TYPE "UDT_RIOVSUStatus"
VERSION : 0.1
   STRUCT
      PNSlaveNotOnline { ExternalAccessible := 'False'; ExternalVisible := 'False'; ExternalWritable := 'False'} : Bool;   // Profinet slave is not online
      PNSlaveError { ExternalAccessible := 'False'; ExternalVisible := 'False'; ExternalWritable := 'False'} : Bool;   // Profinet slave has an error
      "400VCircuitBreaker" { ExternalAccessible := 'False'; ExternalVisible := 'False'; ExternalWritable := 'False'} : Bool;   // 400V Circuit breaker has tripped
      BrakeCircuitBreaker { ExternalAccessible := 'False'; ExternalVisible := 'False'; ExternalWritable := 'False'} : Bool;   // Brake Circuit breaker has tripped
      BrakeThermalError { ExternalAccessible := 'False'; ExternalVisible := 'False'; ExternalWritable := 'False'} : Bool;   // Brake of the servo unit is giving a thermal error
      "24VPowersupplyError" { ExternalAccessible := 'False'; ExternalVisible := 'False'; ExternalWritable := 'False'} : Bool;   // 24V power supply is in error
      ET200sp_ErrorModule : Array[0..31] of Bool;   // True = ET200sp Module has an error or is offline
      PNSlaveWarning { ExternalAccessible := 'False'; ExternalVisible := 'False'; ExternalWritable := 'False'} : Bool;   // Profinet slave has a warning
   END_STRUCT;

END_TYPE

TYPE "UDT_VSUInterface"
TITLE = UDT_VSUInterface
VERSION : 0.1
//User-defined structure of VSU interface parameters.
   STRUCT
      Decisionpoint : Int;   // Point in tracking where the destination is found on the VSU conveyor [mm]
      RequestedPosition : Int;   // Position Requested by destination block
      PositionSetpoint : Int;   // Position number (as configured) to go to by positioning device
      PositionActual : Int;   // Position number the positioning device is actually on
      SwitchingTime : UInt;   // Time it takes to go from one position to the next [ms]
      VSUMainPowerOk { ExternalAccessible := 'False'; ExternalVisible := 'False'; ExternalWritable := 'False'} : Bool;   // True = Main power for VSU ok
      BrakeOk { ExternalAccessible := 'False'; ExternalVisible := 'False'; ExternalWritable := 'False'} : Bool;   // True = VSU brake is ok
      PNDeviceOk { ExternalAccessible := 'False'; ExternalVisible := 'False'; ExternalWritable := 'False'} : Bool;   // Device ok
      Automatic { ExternalAccessible := 'False'; ExternalVisible := 'False'; ExternalWritable := 'False'} : Bool;   // Automatic mode request
      RunEnabled { ExternalAccessible := 'False'; ExternalVisible := 'False'; ExternalWritable := 'False'} : Bool;   // Running of the positioning device is enabled by VSU
      GoReference { ExternalAccessible := 'False'; ExternalVisible := 'False'; ExternalWritable := 'False'} : Bool;   // Activate reference run by VSU
      Referenced { ExternalAccessible := 'False'; ExternalVisible := 'False'; ExternalWritable := 'False'} : Bool;   // Positioning device is referenced
      Manual { ExternalAccessible := 'False'; ExternalVisible := 'False'; ExternalWritable := 'False'} : Bool;   // Manual mode request
      Reference_command { ExternalAccessible := 'False'; ExternalVisible := 'False'; ExternalWritable := 'False'} : Bool;   // Refference command
      JogUp { ExternalAccessible := 'False'; ExternalVisible := 'False'; ExternalWritable := 'False'} : Bool;   // Jog request to move equipment up
      JogDown { ExternalAccessible := 'False'; ExternalVisible := 'False'; ExternalWritable := 'False'} : Bool;   // Jog request to move equipment down
      Ready { ExternalAccessible := 'False'; ExternalVisible := 'False'; ExternalWritable := 'False'} : Bool;   // Positioning block is running and error free
      MotorRunning { ExternalAccessible := 'False'; ExternalVisible := 'False'; ExternalWritable := 'False'} : Bool;   // Motor is running
      Positioning { ExternalAccessible := 'False'; ExternalVisible := 'False'; ExternalWritable := 'False'} : Bool;   // positioning device is moving to its position
      ResetStatistics { ExternalAccessible := 'False'; ExternalVisible := 'False'; ExternalWritable := 'False'} : Bool;   // Reset statistics
      InternalErrorRIOPanel { ExternalAccessible := 'False'; ExternalVisible := 'False'; ExternalWritable := 'False'} : Bool;   // RIO panel has an internal error
      InternalWarningRIOPanel { ExternalAccessible := 'False'; ExternalVisible := 'False'; ExternalWritable := 'False'} : Bool;   // RIO panel has an internal waring
      InternalErrorVFD { ExternalAccessible := 'False'; ExternalVisible := 'False'; ExternalWritable := 'False'} : Bool;   // positioning device internal error
      InternalWarningVFD { ExternalAccessible := 'False'; ExternalVisible := 'False'; ExternalWritable := 'False'} : Bool;   // positioning device has a warning
      InternalErrorReset { ExternalAccessible := 'False'; ExternalVisible := 'False'; ExternalWritable := 'False'} : Bool;   // Reset internal faults
      StartLowSpeed { ExternalAccessible := 'False'; ExternalVisible := 'False'; ExternalWritable := 'False'} : Bool;   // Positioning device starting in low speed
      RequestDieBackUpstream { ExternalAccessible := 'False'; ExternalVisible := 'False'; ExternalWritable := 'False'} : Bool;   // External request die back to the upstream conveyor of the VSU
      ExternalHold { ExternalAccessible := 'False'; ExternalVisible := 'False'; ExternalWritable := 'False'} : Bool;   // External request to stop the VSU conveyor
   END_STRUCT;

END_TYPE

TYPE "UDT_VfdPositioningStatus"
TITLE = UDT_VfdPositioningStatus
VERSION : 0.1
//User-defined structure of VFD SEW positioning status.
   STRUCT
      ErrorCode : Int;   // Error code
      SubErrorCode : Int;   // Sub error code
      PNSlaveNotOnline : Bool := FALSE;   // Profinet slave is not on line
      PNSlaveError : Bool := FALSE;   // Profinet slave has an error
      InternalError : Bool := FALSE;   // A VFD internal error is active, see error code
      InternalWarning : Bool := FALSE;   // A VFD internal warning is active, see error code
      CommunicationErrorMovikit : Bool := FALSE;   // Communication error with MoviKit
      PositioningTimeOutError : Bool := FALSE;   // Exceeded time to reach position
      PNSlaveWarning { ExternalAccessible := 'False'; ExternalVisible := 'False'; ExternalWritable := 'False'} : Bool;   // Profinet slave has a warning
   END_STRUCT;

END_TYPE

TYPE "UDT_VSULiftStatistics"
TITLE = UDT_VSUStatistics
VERSION : 0.1
//User-defined structure of FB_VerticalSwitch function block statistics.
   STRUCT
      UpTime { ExternalWritable := 'False'} : "UDT_EventStatistic";   // VSU up time
      DownTime { ExternalWritable := 'False'} : "UDT_EventStatistic";   // VSU down time
      ExitGapErr { ExternalWritable := 'False'} : "UDT_EventStatistic";   // Error statistics for VSU
      EntryGapErr { ExternalWritable := 'False'} : "UDT_EventStatistic";   // Error statistics for VSU
      BeltTear1Err { ExternalWritable := 'False'} : "UDT_EventStatistic";   // Error statistics for VSU
      BeltTear2Err { ExternalWritable := 'False'} : "UDT_EventStatistic";   // Error statistics for VSU
      MaintSupport1Err { ExternalWritable := 'False'} : "UDT_EventStatistic";   // Error statistics for VSU
      MaintSupport2Err { ExternalWritable := 'False'} : "UDT_EventStatistic";   // Error statistics for VSU
      UpperPositionErr { ExternalWritable := 'False'} : "UDT_EventStatistic";   // Error statistics for VSU
      LowerPositionErr { ExternalWritable := 'False'} : "UDT_EventStatistic";   // Error statistics for VSU
      SafetyDoorErr { ExternalWritable := 'False'} : "UDT_EventStatistic";   // Error statistics for VSU
      Direction_Error { ExternalWritable := 'False'} : "UDT_EventStatistic";   // Error statistics for VSU
   END_STRUCT;

END_TYPE

TYPE "UDT_VfdPositioningConfiguration"
TITLE = UDT_VfdPositioningConfiguration
VERSION : 0.1
//User defined stucture for configuring positioning device
   STRUCT
      TorqueMax : Real;   // VFD torque max - reference [Nm] as set up in SEW project
      SupplyFdbckOnDelayTime : UDInt;   // On delay time for supply feedback [ms]
      PositionWindow : DInt;   // Position window (tolerance) [mm]
      PositionMax : DInt;   // Maximum allowed position [mm]
      PositionMin : DInt;   // Minimum allowed position [mm]
      VFDSpeed : Int;   // Speed to run in automatic mode [mm/s]
      VFDAccDecel : Int;   // Acceleration and deceleration [mm/s2]
      VFDPNDeviceName : String;   // VFD's device name
      Position : Array[0..10] of DInt;   // Positions in mm to move to as requested
   END_STRUCT;

END_TYPE

TYPE "UDT_VfdSEWSpeedPO"
TITLE = UDT_VFD_SEW_PO
VERSION : 0.1
//User-defined structure of VFD SEW output telegram.
   STRUCT
      Control_Word_1 : Struct   // Control Word 1
         ResetError { ExternalAccessible := 'False'; ExternalVisible := 'False'; ExternalWritable := 'False'} : Bool;   // Reset error "1"
         BIT_09_Reserved { ExternalAccessible := 'False'; ExternalVisible := 'False'; ExternalWritable := 'False'} : Bool;   // Reserved
         ActivateDriveTrain2 { ExternalAccessible := 'False'; ExternalVisible := 'False'; ExternalWritable := 'False'} : Bool;   // Activate drive train 2 "1"
         BIT_11_Reserved { ExternalAccessible := 'False'; ExternalVisible := 'False'; ExternalWritable := 'False'} : Bool;   // Reserved
         DeactivateSW_LimitSwitch { ExternalAccessible := 'False'; ExternalVisible := 'False'; ExternalWritable := 'False'} : Bool;   // Deactivate software limit switch "1"
         ActivateInhibit { ExternalAccessible := 'False'; ExternalVisible := 'False'; ExternalWritable := 'False'} : Bool;   // Activate inhibit "1"
         ActivateStandby { ExternalAccessible := 'False'; ExternalVisible := 'False'; ExternalWritable := 'False'} : Bool;   // Activate standby "1"
         MovikitHandshakeIn { ExternalAccessible := 'False'; ExternalVisible := 'False'; ExternalWritable := 'False'} : Bool;   // If the MOVIKIT works the value will be copied into "MovikitHandshakeOut"
         EnableRapidStop { ExternalAccessible := 'False'; ExternalVisible := 'False'; ExternalWritable := 'False'} : Bool;   // Enable “1” / Rapid stop “0”
         EnableApplicationStop { ExternalAccessible := 'False'; ExternalVisible := 'False'; ExternalWritable := 'False'} : Bool;   // Enable “1” / Application stop “0”
         BIT_02_Reserved { ExternalAccessible := 'False'; ExternalVisible := 'False'; ExternalWritable := 'False'} : Bool;   // Reserved
         ReleaseBrake { ExternalAccessible := 'False'; ExternalVisible := 'False'; ExternalWritable := 'False'} : Bool;   // Release brake "1"
         JogPos { ExternalAccessible := 'False'; ExternalVisible := 'False'; ExternalWritable := 'False'} : Bool;   // Jog in positive direction "1"
         JogNeg { ExternalAccessible := 'False'; ExternalVisible := 'False'; ExternalWritable := 'False'} : Bool;   // Jog in negative direction "1"
         ApplyRelativePositioning { ExternalAccessible := 'False'; ExternalVisible := 'False'; ExternalWritable := 'False'} : Bool;   // Take the relative position from the FCB09 "1"
         StartStop { ExternalAccessible := 'False'; ExternalVisible := 'False'; ExternalWritable := 'False'} : Bool;   // Start "1" / Stop "0"
      END_STRUCT;
      SetpointSpeed : Int;   // Speed (Int) in rpm
      SetpointAcceleration : Int;   // Acceleration (Int) in rpm/s
      SetpointDeceleration : Int;   // Decceleration (Int) in rpm/s
   END_STRUCT;

END_TYPE

TYPE "UDT_AixPlcFullControllerConfiguration"
TITLE = UDT_VFD_Configuration
VERSION : 0.1
//User-defined structure oparameters.
   STRUCT
      AixContrlPNDeviceName { ExternalAccessible := 'False'; ExternalVisible := 'False'; ExternalWritable := 'False'} : String;   // Ai2's Controller Profinet device name
      Motor { ExternalAccessible := 'False'; ExternalVisible := 'False'; ExternalWritable := 'False'} : Struct
         RampUpTime { ExternalAccessible := 'False'; ExternalVisible := 'False'; ExternalWritable := 'False'} : UDInt := 100;   // Ramp up time for monitoring starting [ms]
         RampDownTime { ExternalAccessible := 'False'; ExternalVisible := 'False'; ExternalWritable := 'False'} : UDInt := 100;   // Ramp up time for monitoring stopping [ms]
         SpeedSetpointWindow { ExternalAccessible := 'False'; ExternalVisible := 'False'; ExternalWritable := 'False'} : Int := 5;   // Speed setpoint window (tolerance) [mm/s]
         Ratio { ExternalAccessible := 'False'; ExternalVisible := 'False'; ExternalWritable := 'False'} : Real := 1.0;   // Ratio conveyor roller to driven roller
         DirectionReversal { ExternalAccessible := 'False'; ExternalVisible := 'False'; ExternalWritable := 'False'} : Bool;   // True = direction will be reversed
         InterlockFwd { ExternalAccessible := 'False'; ExternalVisible := 'False'; ExternalWritable := 'False'} : Bool := TRUE;   // False = running in forward direction is not possible / allowed
         InterlockRvs { ExternalAccessible := 'False'; ExternalVisible := 'False'; ExternalWritable := 'False'} : Bool;   // False = running in reverse direction is not possible / allowed
         MotorExist { ExternalAccessible := 'False'; ExternalVisible := 'False'; ExternalWritable := 'False'} : Bool;   // True = Motor output connected
      END_STRUCT;
   END_STRUCT;

END_TYPE

TYPE "UDT_AixPlcFullIn"
VERSION : 0.1
   STRUCT
      ConveyStopStatus { ExternalVisible := 'False'} : Struct   // Status of ConveyStop
         Bit08 { ExternalAccessible := 'False'; ExternalVisible := 'False'; ExternalWritable := 'False'} : Bool;   // Reserved
         Bit09 { ExternalAccessible := 'False'; ExternalVisible := 'False'; ExternalWritable := 'False'} : Bool;   // Reserved
         StopActiveCommandPLC { ExternalAccessible := 'False'; ExternalVisible := 'False'; ExternalWritable := 'False'} : Bool;   // Stop active due to stop command from the PLC
         Bit11 { ExternalAccessible := 'False'; ExternalVisible := 'False'; ExternalWritable := 'False'} : Bool;   // Reserved
         Bit12 { ExternalAccessible := 'False'; ExternalVisible := 'False'; ExternalWritable := 'False'} : Bool;   // Reserved
         Bit13 { ExternalAccessible := 'False'; ExternalVisible := 'False'; ExternalWritable := 'False'} : Bool;   // Reserved
         Bit14 { ExternalAccessible := 'False'; ExternalVisible := 'False'; ExternalWritable := 'False'} : Bool;   // Reserved
         Bit15 { ExternalAccessible := 'False'; ExternalVisible := 'False'; ExternalWritable := 'False'} : Bool;   // Reserved
         Bit00 { ExternalAccessible := 'False'; ExternalVisible := 'False'; ExternalWritable := 'False'} : Bool;   // Reserved
         Bit01 { ExternalAccessible := 'False'; ExternalVisible := 'False'; ExternalWritable := 'False'} : Bool;   // Reserved
         Bit02 { ExternalAccessible := 'False'; ExternalVisible := 'False'; ExternalWritable := 'False'} : Bool;   // Reserved
         Bit03 { ExternalAccessible := 'False'; ExternalVisible := 'False'; ExternalWritable := 'False'} : Bool;   // Reserved
         Bit04 { ExternalAccessible := 'False'; ExternalVisible := 'False'; ExternalWritable := 'False'} : Bool;   // Reserved
         StopActiveOtherModule { ExternalAccessible := 'False'; ExternalVisible := 'False'; ExternalWritable := 'False'} : Bool;   // Stop condition is active on a module in the ConveyStop group
         StopActiveLostConn { ExternalAccessible := 'False'; ExternalVisible := 'False'; ExternalWritable := 'False'} : Bool;   // Stop is active due to a loss of communication connection
         StopActiveLostPLC { ExternalAccessible := 'False'; ExternalVisible := 'False'; ExternalWritable := 'False'} : Bool;   // Stop active due to a loss of connection with the PLC
      END_STRUCT;
      AllSensorPortInputs { ExternalVisible := 'False'} : Struct   // Left and Right Sensor Port inputs
         Bit08 { ExternalAccessible := 'False'; ExternalVisible := 'False'; ExternalWritable := 'False'} : Bool;   // Reserved
         Bit09 { ExternalAccessible := 'False'; ExternalVisible := 'False'; ExternalWritable := 'False'} : Bool;   // Reserved
         Bit10 { ExternalAccessible := 'False'; ExternalVisible := 'False'; ExternalWritable := 'False'} : Bool;   // Reserved
         Bit11 { ExternalAccessible := 'False'; ExternalVisible := 'False'; ExternalWritable := 'False'} : Bool;   // Reserved
         Bit12 { ExternalAccessible := 'False'; ExternalVisible := 'False'; ExternalWritable := 'False'} : Bool;   // Reserved
         Bit13 { ExternalAccessible := 'False'; ExternalVisible := 'False'; ExternalWritable := 'False'} : Bool;   // Reserved
         Bit14 { ExternalAccessible := 'False'; ExternalVisible := 'False'; ExternalWritable := 'False'} : Bool;   // Reserved
         Heartbeat { ExternalAccessible := 'False'; ExternalVisible := 'False'; ExternalWritable := 'False'} : Bool;   // This bit toggles every 2 seconds
         LeftPin2 { ExternalAccessible := 'False'; ExternalVisible := 'False'; ExternalWritable := 'False'} : Bool;   // Left sensor port Pin2 state
         Bit01 { ExternalAccessible := 'False'; ExternalVisible := 'False'; ExternalWritable := 'False'} : Bool;   // Reserved
         RightPin2 { ExternalAccessible := 'False'; ExternalVisible := 'False'; ExternalWritable := 'False'} : Bool;   // Right sensor port Pin2 state
         Bit03 { ExternalAccessible := 'False'; ExternalVisible := 'False'; ExternalWritable := 'False'} : Bool;   // Reserved
         LeftSensor { ExternalAccessible := 'False'; ExternalVisible := 'False'; ExternalWritable := 'False'} : Bool;   // Left sensor port Pin4 state
         Bit05 { ExternalAccessible := 'False'; ExternalVisible := 'False'; ExternalWritable := 'False'} : Bool;   // Reserved
         RightSensor { ExternalAccessible := 'False'; ExternalVisible := 'False'; ExternalWritable := 'False'} : Bool;   // Right sensor port Pin4 state
         Bit07 { ExternalAccessible := 'False'; ExternalVisible := 'False'; ExternalWritable := 'False'} : Bool;   // Reserved
      END_STRUCT;
      SensorDetect { ExternalVisible := 'False'} : Struct   // Sensor detection
         Bits08_15 { ExternalVisible := 'False'} : SInt;   // Reserved
         RightSensorDetect { ExternalAccessible := 'False'; ExternalVisible := 'False'; ExternalWritable := 'False'} : Bool;   // True when sensor is detected
         LeftSensorDetect { ExternalAccessible := 'False'; ExternalVisible := 'False'; ExternalWritable := 'False'} : Bool;   // True when sensor is detected
         Bit02 { ExternalAccessible := 'False'; ExternalVisible := 'False'; ExternalWritable := 'False'} : Bool;   // Reserved
         Bit03 { ExternalAccessible := 'False'; ExternalVisible := 'False'; ExternalWritable := 'False'} : Bool;   // Reserved
         Bit04 { ExternalAccessible := 'False'; ExternalVisible := 'False'; ExternalWritable := 'False'} : Bool;   // Reserved
         Bit05 { ExternalAccessible := 'False'; ExternalVisible := 'False'; ExternalWritable := 'False'} : Bool;   // Reserved
         Bit06 { ExternalAccessible := 'False'; ExternalVisible := 'False'; ExternalWritable := 'False'} : Bool;   // Reserved
         Bit07 { ExternalAccessible := 'False'; ExternalVisible := 'False'; ExternalWritable := 'False'} : Bool;   // Reserved
      END_STRUCT;
      VoltageMotors { ExternalVisible := 'False'} : Int;   // The Voltage applied to the module's motor power connection in millivolts
      LeftMotorCurrent { ExternalVisible := 'False'} : Int;   // Left motor running current in milliamperes
      LeftMotorFreq { ExternalVisible := 'False'} : Int;   // Left motor running electrical frequency in Hz
      LeftMotorCalcTemp { ExternalVisible := 'False'} : Byte;   // Left motor temperature in degrees C
      ModuleTemp { ExternalVisible := 'False'} : Byte;   // Module CPU temperature in degrees C
      LeftMotorDiagnostic { ExternalVisible := 'False'} : Struct   // Left motor diagnostics .
         Overheat { ExternalAccessible := 'False'; ExternalVisible := 'False'; ExternalWritable := 'False'} : Bool;   // Left motor temperature has exceeded 105 degrees Celsius
         MaxTorque { ExternalAccessible := 'False'; ExternalVisible := 'False'; ExternalWritable := 'False'} : Bool;   // Left motor at maximum torque output
         ShortCircuit { ExternalAccessible := 'False'; ExternalVisible := 'False'; ExternalWritable := 'False'} : Bool;   // Left motor short circuit
         MotorNotConnected { ExternalAccessible := 'False'; ExternalVisible := 'False'; ExternalWritable := 'False'} : Bool;   // Left motor is not connected
         Overload { ExternalAccessible := 'False'; ExternalVisible := 'False'; ExternalWritable := 'False'} : Bool;   // Left motor overloaded after more than 20 seconds in Stalled
         Stalled { ExternalAccessible := 'False'; ExternalVisible := 'False'; ExternalWritable := 'False'} : Bool;   // Left motor stalled and speed is less than 10% of the set speed
         BadHall { ExternalAccessible := 'False'; ExternalVisible := 'False'; ExternalWritable := 'False'} : Bool;   // Left motor Hall Effect Sensor error active
         MotorNotUsed { ExternalAccessible := 'False'; ExternalVisible := 'False'; ExternalWritable := 'False'} : Bool;   // Left motor not used
         MotorStatus1 { ExternalAccessible := 'False'; ExternalVisible := 'False'; ExternalWritable := 'False'} : Bool;   // Left motor running and direction status
         MotorStatus2 { ExternalAccessible := 'False'; ExternalVisible := 'False'; ExternalWritable := 'False'} : Bool;   // Left motor running and direction status
         MotorPortinDOmode { ExternalAccessible := 'False'; ExternalVisible := 'False'; ExternalWritable := 'False'} : Bool;   // Left motor port is in digital Output mode .
         ReservedBit03 { ExternalAccessible := 'False'; ExternalVisible := 'False'; ExternalWritable := 'False'} : Bool;   // Reserved
         ReservedBit04 { ExternalAccessible := 'False'; ExternalVisible := 'False'; ExternalWritable := 'False'} : Bool;   // Reserved
         BoardOverheat { ExternalAccessible := 'False'; ExternalVisible := 'False'; ExternalWritable := 'False'} : Bool;   // Board temperature has exceeded 90 degrees Celsius
         OverVoltage { ExternalAccessible := 'False'; ExternalVisible := 'False'; ExternalWritable := 'False'} : Bool;   // Supply voltage + motor back EMF exceeded 30 volts
         LowVoltage { ExternalAccessible := 'False'; ExternalVisible := 'False'; ExternalWritable := 'False'} : Bool;   // Module power supply is less than 18 Volts
      END_STRUCT;
      RightMotorCurrent { ExternalVisible := 'False'} : Int;   // Right motor running current in milliamperes
      RightMotorFreq { ExternalVisible := 'False'} : Int;   // Right motor running electrical frequency in Hz
      RightMotorCalcTemp { ExternalVisible := 'False'} : Byte;   // Right motor temperature in degrees Celsius
      ModuleTemp1 { ExternalVisible := 'False'} : Byte;   // Module PCB temperature in degrees C (same as ModuleTemp tag)
      RightMotorDiagnostic { ExternalVisible := 'False'} : Struct   // Right motor diagnostics .
         Overheat { ExternalAccessible := 'False'; ExternalVisible := 'False'; ExternalWritable := 'False'} : Bool;   // Right motor temperature has exceeded 105 degrees Celsius
         MaxTorque { ExternalAccessible := 'False'; ExternalVisible := 'False'; ExternalWritable := 'False'} : Bool;   // Right motor at maximum torque output
         ShortCircuit { ExternalAccessible := 'False'; ExternalVisible := 'False'; ExternalWritable := 'False'} : Bool;   // Right motor short circuit
         MotorNotConnected { ExternalAccessible := 'False'; ExternalVisible := 'False'; ExternalWritable := 'False'} : Bool;   // Right motor is not connected
         Overload { ExternalAccessible := 'False'; ExternalVisible := 'False'; ExternalWritable := 'False'} : Bool;   // Right motor overloaded after more than 20 seconds in Stalled
         Stalled { ExternalAccessible := 'False'; ExternalVisible := 'False'; ExternalWritable := 'False'} : Bool;   // Right motor stalled and speed is less than 10% of the set speed
         BadHall { ExternalAccessible := 'False'; ExternalVisible := 'False'; ExternalWritable := 'False'} : Bool;   // Right motor Hall Effect Sensor error active
         MotorNotUsed { ExternalAccessible := 'False'; ExternalVisible := 'False'; ExternalWritable := 'False'} : Bool;   // Right motor is not used
         MotorStatus1 { ExternalAccessible := 'False'; ExternalVisible := 'False'; ExternalWritable := 'False'} : Bool;   // Right motor running and direction status
         MotorStatus2 { ExternalAccessible := 'False'; ExternalVisible := 'False'; ExternalWritable := 'False'} : Bool;   // Right motor running and direction status
         MotorPortinDOmode { ExternalAccessible := 'False'; ExternalVisible := 'False'; ExternalWritable := 'False'} : Bool;   // Right motor port is in digital output mode .
         ReservedBit03 { ExternalAccessible := 'False'; ExternalVisible := 'False'; ExternalWritable := 'False'} : Bool;   // Reserved
         ReservedBit04 { ExternalAccessible := 'False'; ExternalVisible := 'False'; ExternalWritable := 'False'} : Bool;   // Reserved
         BoardOverheat { ExternalAccessible := 'False'; ExternalVisible := 'False'; ExternalWritable := 'False'} : Bool;   // Board temperature has exceeded 90 degrees Celsius
         OverVoltage { ExternalAccessible := 'False'; ExternalVisible := 'False'; ExternalWritable := 'False'} : Bool;   // Supply voltage + motor back EMF exceeded 30 volts
         LowVoltage { ExternalAccessible := 'False'; ExternalVisible := 'False'; ExternalWritable := 'False'} : Bool;   // Module power supply is less than 18 Volts
      END_STRUCT;
      LeftMotorDIOstatus { ExternalVisible := 'False'} : Struct   // Status of Left M8 motor port when used as a digital IO
         Bit08 { ExternalAccessible := 'False'; ExternalVisible := 'False'; ExternalWritable := 'False'} : Bool;   // Reserved
         Bit09 { ExternalAccessible := 'False'; ExternalVisible := 'False'; ExternalWritable := 'False'} : Bool;   // Reserved
         Bit10 { ExternalAccessible := 'False'; ExternalVisible := 'False'; ExternalWritable := 'False'} : Bool;   // Reserved
         Bit11 { ExternalAccessible := 'False'; ExternalVisible := 'False'; ExternalWritable := 'False'} : Bool;   // Reserved
         ShortCircuit { ExternalAccessible := 'False'; ExternalVisible := 'False'; ExternalWritable := 'False'} : Bool;   // Short circuit between +24V and any of the U,V,W phases
         Bit13 { ExternalAccessible := 'False'; ExternalVisible := 'False'; ExternalWritable := 'False'} : Bool;   // Reserved
         Bit14 { ExternalAccessible := 'False'; ExternalVisible := 'False'; ExternalWritable := 'False'} : Bool;   // Reserved
         Bit15 { ExternalAccessible := 'False'; ExternalVisible := 'False'; ExternalWritable := 'False'} : Bool;   // Reserved
         Bits00_07 { ExternalVisible := 'False'} : SInt;   // Reserved
      END_STRUCT;
      RightMotorDIOstatus { ExternalVisible := 'False'} : Struct   // Status of Right M8 motor port when used as a digital IO
         Bit08 { ExternalAccessible := 'False'; ExternalVisible := 'False'; ExternalWritable := 'False'} : Bool;   // Reserved
         Bit09 { ExternalAccessible := 'False'; ExternalVisible := 'False'; ExternalWritable := 'False'} : Bool;   // Reserved
         Bit10 { ExternalAccessible := 'False'; ExternalVisible := 'False'; ExternalWritable := 'False'} : Bool;   // Reserved
         Bit11 { ExternalAccessible := 'False'; ExternalVisible := 'False'; ExternalWritable := 'False'} : Bool;   // Reserved
         ShortCircuit { ExternalAccessible := 'False'; ExternalVisible := 'False'; ExternalWritable := 'False'} : Bool;   // Short circuit between +24V and any of the U,V,W phases
         Bit13 { ExternalAccessible := 'False'; ExternalVisible := 'False'; ExternalWritable := 'False'} : Bool;   // Reserved
         Bit14 { ExternalAccessible := 'False'; ExternalVisible := 'False'; ExternalWritable := 'False'} : Bool;   // Reserved
         Bit15 { ExternalAccessible := 'False'; ExternalVisible := 'False'; ExternalWritable := 'False'} : Bool;   // Reserved
         Bits00_07 { ExternalVisible := 'False'} : SInt;   // Reserved
      END_STRUCT;
      UpstreamModuleStatus { ExternalVisible := 'False'} : Word;   // The ZPA status from the Upstream ConveyLinx module
      DownstreamModuleStatus { ExternalVisible := 'False'} : Word;   // The ZPA status from the Downstream ConveyLinx module
      TrackingFromUpstream { ExternalVisible := 'False'} : DWord;   // Tracking data from the Upstream ConveyLinx module
      Index18 { ExternalVisible := 'False'} : Word;   // Index
      ServoLocationLeft { ExternalVisible := 'False'} : Int;   // Left motor current location from 0 in mm for MDR and in pulses for PGD
      ServoLocationRight { ExternalVisible := 'False'} : Int;   // Right motor current location from 0 in mm for MDR and in pulses for PGD
      ServoStatusLeft { ExternalVisible := 'False'} : Word;   // Left motor servo commands status
      ServoStatusRight { ExternalVisible := 'False'} : Word;   // Right motor servo commands status
      LeftMotorActualSpeed { ExternalVisible := 'False'} : Word;   // Bits 0 thru 13: Left motor actual speed in mm/sec, Bits 14-15: Status. For PGD, base unit is 1/10 RPM
      RightMotorActualSpeed { ExternalVisible := 'False'} : Word;   // Bits 0 thru 13: Left motor actual speed in mm/sec, Bits 14-15: Status. For PGD, base unit is 1/10 RPM
      Future { ExternalVisible := 'False'} : Array[25..31] of Int;   // Future
   END_STRUCT;

END_TYPE

TYPE "UDT_VfdSEWSpeedPI"
TITLE = UDT_VFD_SEW_PI
VERSION : 0.1
//User-defined structure of VFD SEW input telegram.
   STRUCT
      Status_Word_1 : Struct   // Status Word 1
         Error { ExternalAccessible := 'False'; ExternalVisible := 'False'; ExternalWritable := 'False'} : Bool;   // An error is active "1"
         Warning { ExternalAccessible := 'False'; ExternalVisible := 'False'; ExternalWritable := 'False'} : Bool;   // A warning is active "1"
         DriveTrain2Active { ExternalAccessible := 'False'; ExternalVisible := 'False'; ExternalWritable := 'False'} : Bool;   // Drive train 2 is active "1"
         VelocityTargetActualComparison { ExternalAccessible := 'False'; ExternalVisible := 'False'; ExternalWritable := 'False'} : Bool;   // The notification "Velocity target-actual-comparison" is on "1"
         SW_LimitSwitchInactive { ExternalAccessible := 'False'; ExternalVisible := 'False'; ExternalWritable := 'False'} : Bool;   // he software limit switch is inactive "1"
         BIT_13_Reserved { ExternalAccessible := 'False'; ExternalVisible := 'False'; ExternalWritable := 'False'} : Bool;   // Reserved
         StandbyActive { ExternalAccessible := 'False'; ExternalVisible := 'False'; ExternalWritable := 'False'} : Bool;   // Standby mode is active "1"
         MovikitHandshakeOut { ExternalAccessible := 'False'; ExternalVisible := 'False'; ExternalWritable := 'False'} : Bool;   // Copied value of "MovikitHandshakeIn"
         InverterReady { ExternalAccessible := 'False'; ExternalVisible := 'False'; ExternalWritable := 'False'} : Bool;   // There's no error and the inverter is ready "1"
         STO_Inactive { ExternalAccessible := 'False'; ExternalVisible := 'False'; ExternalWritable := 'False'} : Bool;   // STO is not active "1"
         OutputStageEnabled { ExternalAccessible := 'False'; ExternalVisible := 'False'; ExternalWritable := 'False'} : Bool;   // The output stage is released "1"
         BrakeReleased { ExternalAccessible := 'False'; ExternalVisible := 'False'; ExternalWritable := 'False'} : Bool;   // The brake is released "1"
         DriveActive { ExternalAccessible := 'False'; ExternalVisible := 'False'; ExternalWritable := 'False'} : Bool;   // The drive is active and the shaft turning "1"
         Referenced { ExternalAccessible := 'False'; ExternalVisible := 'False'; ExternalWritable := 'False'} : Bool;   // The drive is referenced "1"
         RelativePositionApplied { ExternalAccessible := 'False'; ExternalVisible := 'False'; ExternalWritable := 'False'} : Bool;   // The relative position is applied "1"
         InPosition { ExternalAccessible := 'False'; ExternalVisible := 'False'; ExternalWritable := 'False'} : Bool;   // The notification "in position" is on "1"
      END_STRUCT;
      ActualSpeed : Int;   // Actual drive speed (Int) in rpm
      StatusErrorNo : Word;   // Current status of the drive
      ActualTorque : Int;   // Actual torque in percent od the rated unit torque
   END_STRUCT;

END_TYPE

TYPE "UDT_StatisticsTC13"
VERSION : 0.1
//One direction, motor, EoS, Tracking
   STRUCT
      Conveyor : "UDT_ConveyorStatistics";   // Conveyor Statistics
      PEC_EoS : "UDT_PECUpdateStatistics";   // PEC EoS Statistics
      MCO_M01 : "UDT_VfdStatistics";   // MCO Statistics
   END_STRUCT;

END_TYPE

TYPE "UDT_StatisticsTC07"
VERSION : 0.1
//One direction, motor, controler, EoS, Stop blade
   STRUCT
      Conveyor : "UDT_ConveyorStatistics";   // Conveyor Statistics
      PEC_EoS : "UDT_PECStatistics";   // PEC EoS Statistics
      MCO_M01 : "UDT_VfdStatistics";   // MCO Statistics
      BladeStopEoS : "UDT_ValveStatistics";   // Blade stop EoS statistics
   END_STRUCT;

END_TYPE

TYPE "UDT_StatisticsTC02"
VERSION : 0.1
//One direction, motor, controler, EoS
   STRUCT
      Conveyor : "UDT_ConveyorStatistics";   // Conveyor Statistics
      PEC_EoS : "UDT_PECStatistics";   // PEC EoS Statistics
      MCO_M01 : "UDT_VfdStatistics";   // MCO Statistics
   END_STRUCT;

END_TYPE

TYPE "UDT_StatisticsTC03"
VERSION : 0.1
//One direction, motor, controler, EoS, Tracking
   STRUCT
      Conveyor : "UDT_ConveyorStatistics";   // Conveyor Statistics
      PEC_EoS : "UDT_PECUpdateStatistics";   // PEC EoS Statistics
      MCO_M01 : "UDT_VfdStatistics";   // MCO Statistics
   END_STRUCT;

END_TYPE

TYPE "UDT_HMICommandTC36"
VERSION : 0.1
//One direction, motor, controler
   STRUCT
      RightAngledTransfer : "UDT_RATCommand";   // Conveyor Statistics
   END_STRUCT;

END_TYPE

TYPE "UDT_HMICommandTCxx"
VERSION : 0.1
//One direction, motor, controler
   STRUCT
      Conveyor : "UDT_ConveyorCommand";   // Conveyor Statistics
   END_STRUCT;

END_TYPE

TYPE "UDT_RATConfiguration"
VERSION : 0.1
   STRUCT
      OutfeedTimeDelay { ExternalAccessible := 'False'; ExternalVisible := 'False'; ExternalWritable := 'False'} : UDInt;   // PEC on delaytime
      InfeedTimeDelay { ExternalAccessible := 'False'; ExternalVisible := 'False'; ExternalWritable := 'False'} : UDInt;   // PEC off delaytime
      SectionUpMonitoringTime { ExternalAccessible := 'False'; ExternalVisible := 'False'; ExternalWritable := 'False'} : UDInt := 500;   // Runtime delay lifting device up signal on delay
      SectionDownMonitoringTime { ExternalAccessible := 'False'; ExternalVisible := 'False'; ExternalWritable := 'False'} : UDInt := 500;   // Runtime delay lifting device down signal on delay
      BladeStopUpMonitoringTime { ExternalAccessible := 'False'; ExternalVisible := 'False'; ExternalWritable := 'False'} : UDInt := 500;   // Runtime delay lifting blade stop up signal on delay
      BladeStopDownMonitoringTime { ExternalAccessible := 'False'; ExternalVisible := 'False'; ExternalWritable := 'False'} : UDInt := 500;   // Runtime delay lifting blade stop down signal on delay
      InfeedADistance { ExternalAccessible := 'False'; ExternalVisible := 'False'; ExternalWritable := 'False'} : Int;   // Distance between A infeed photoeye and place where we want to stop tail of product during infeed [mm]
      InfeedBDistance { ExternalAccessible := 'False'; ExternalVisible := 'False'; ExternalWritable := 'False'} : Int;   // Distance between B infeed photoeye and place where we want to stop tail of product during infeed [mm]
      InfeedCDistance { ExternalAccessible := 'False'; ExternalVisible := 'False'; ExternalWritable := 'False'} : Int;   // Distance between C infeed photoeye and place where we want to stop tail of product during infeed [mm]
      InfeedDDistance { ExternalAccessible := 'False'; ExternalVisible := 'False'; ExternalWritable := 'False'} : Int;   // Distance between D infeed photoeye and place where we want to stop tail of product during infeed [mm]
      InfeedTimeout { ExternalAccessible := 'False'; ExternalVisible := 'False'; ExternalWritable := 'False'} : UDInt := 60000;   // The time after which an error is triggered when a package is not received [ms]
      ReactivationTime { ExternalAccessible := 'False'; ExternalVisible := 'False'; ExternalWritable := 'False'} : UDInt := 30000;   // After this time RAT will be restarted if hang [ms]
      DefaultPosition { ExternalAccessible := 'False'; ExternalVisible := 'False'; ExternalWritable := 'False'} : Int;   // 0 = dont care, 1 = go down after, 2 = go up after
      DefaultDestination { ExternalAccessible := 'False'; ExternalVisible := 'False'; ExternalWritable := 'False'} : Int;   // 1 = upstream conveyor default, 2 = downstream conveyor default, 3 = right conveyor default, 4 = left conveyor default, 0= wait until destination is received
      ConveyorADestination { ExternalAccessible := 'False'; ExternalVisible := 'False'; ExternalWritable := 'False'} : Int;   // Unique Conveyor A outfeed destination number
      ConveyorBDestination { ExternalAccessible := 'False'; ExternalVisible := 'False'; ExternalWritable := 'False'} : Int;   // Unique Conveyor B outfeed destination number
      ConveyorCDestination { ExternalAccessible := 'False'; ExternalVisible := 'False'; ExternalWritable := 'False'} : Int;   // Unique Conveyor C outfeed destination number
      ConveyorDDestination { ExternalAccessible := 'False'; ExternalVisible := 'False'; ExternalWritable := 'False'} : Int;   // Unique Conveyor D outfeed destination number
      ControlProductWithPEC { ExternalAccessible := 'False'; ExternalVisible := 'False'; ExternalWritable := 'False'} : Bool := TRUE;   // TRUE when product presence should be checked by the diagonal PEC
      BladeStopEoS { ExternalAccessible := 'False'; ExternalVisible := 'False'; ExternalWritable := 'False'} : Bool := FALSE;   // TRUE when blade stop at the end of section is present
      BladeStopBoS { ExternalAccessible := 'False'; ExternalVisible := 'False'; ExternalWritable := 'False'} : Bool := FALSE;   // TRUE when blade stop at the beginning of section is present
      PositionVerification { ExternalAccessible := 'False'; ExternalVisible := 'False'; ExternalWritable := 'False'} : Bool := FALSE;   // TRUE when position verification during movement is required
   END_STRUCT;

END_TYPE

TYPE "UDT_VfdSEWPositioningPI"
TITLE = UDT_VfdSEWPositioningPI
VERSION : 0.1
//User-defined structure of VFD SEW input telegram.
   STRUCT
      Status_Word_1 : Struct   // Status Word 1
         Error { ExternalAccessible := 'False'; ExternalVisible := 'False'; ExternalWritable := 'False'} : Bool;   // An error is active "1"
         Warning { ExternalAccessible := 'False'; ExternalVisible := 'False'; ExternalWritable := 'False'} : Bool;   // A warning is active "1"
         DriveTrain2Active { ExternalAccessible := 'False'; ExternalVisible := 'False'; ExternalWritable := 'False'} : Bool;   // Drive train 2 is active "1"
         VelocityTargetActualComparison { ExternalAccessible := 'False'; ExternalVisible := 'False'; ExternalWritable := 'False'} : Bool;   // The notification "Velocity target-actual-comparison" is on "1"
         SW_LimitSwitchInactive { ExternalAccessible := 'False'; ExternalVisible := 'False'; ExternalWritable := 'False'} : Bool;   // he software limit switch is inactive "1"
         BIT_13_Reserved { ExternalAccessible := 'False'; ExternalVisible := 'False'; ExternalWritable := 'False'} : Bool;   // Reserved
         StandbyActive { ExternalAccessible := 'False'; ExternalVisible := 'False'; ExternalWritable := 'False'} : Bool;   // Standby mode is active "1"
         MovikitHandshakeOut { ExternalAccessible := 'False'; ExternalVisible := 'False'; ExternalWritable := 'False'} : Bool;   // Copied value of "MovikitHandshakeIn"
         InverterReady { ExternalAccessible := 'False'; ExternalVisible := 'False'; ExternalWritable := 'False'} : Bool;   // There's no error and the inverter is ready "1"
         STO_Inactive { ExternalAccessible := 'False'; ExternalVisible := 'False'; ExternalWritable := 'False'} : Bool;   // STO is not active "1"
         OutputStageEnabled { ExternalAccessible := 'False'; ExternalVisible := 'False'; ExternalWritable := 'False'} : Bool;   // The output stage is released "1"
         BrakeReleased { ExternalAccessible := 'False'; ExternalVisible := 'False'; ExternalWritable := 'False'} : Bool;   // The brake is released "1"
         DriveActive { ExternalAccessible := 'False'; ExternalVisible := 'False'; ExternalWritable := 'False'} : Bool;   // The drive is active and the shaft turning "1"
         Referenced { ExternalAccessible := 'False'; ExternalVisible := 'False'; ExternalWritable := 'False'} : Bool;   // The drive is referenced "1"
         RelativePositionApplied { ExternalAccessible := 'False'; ExternalVisible := 'False'; ExternalWritable := 'False'} : Bool;   // The relative position is applied "1"
         InPosition { ExternalAccessible := 'False'; ExternalVisible := 'False'; ExternalWritable := 'False'} : Bool;   // The notification "in position" is on "1"
      END_STRUCT;
      ActualSpeed : Int;   // Actual drive speed (Int) [mm/s]
      StatusErrorNo : Word;   // Current status of the drive
      ActualTorque : Int;   // Actual torque in percent od the rated unit torque
      DigitalInput : Word;   // Digital inputs
      Mode : Int;   // Actual application mode (Int)
      ActualPosition_hW : Word;   // Actual position - High Word
      ActualPosition_lW : Word;   // Actual position - Low Word
   END_STRUCT;

END_TYPE

TYPE "UDT_HMICommandTC07"
VERSION : 0.1
//One direction, motor, controler
   STRUCT
      Conveyor { S7_SetPoint := 'False'} : "UDT_ConveyorCommand";   // Conveyor HMI commands
      BladeStopEoS { S7_SetPoint := 'False'} : "UDT_ValveCommand";   // Blade Stop EoS HMI commands
   END_STRUCT;

END_TYPE

TYPE "UDT_VSUCommand"
TITLE = UDT_VSUCommand
VERSION : 0.1
//User-defined structure of VSU commands.
   STRUCT
      SemiAutomaticMode { ExternalAccessible := 'False'; ExternalVisible := 'False'; ExternalWritable := 'False'} : Bool;   // Semiautomatic mode command from HMI
      ManualMode { ExternalAccessible := 'False'; ExternalVisible := 'False'; ExternalWritable := 'False'} : Bool;   // Manual mode command from HMI
      CommandUp { ExternalAccessible := 'False'; ExternalVisible := 'False'; ExternalWritable := 'False'} : Bool;   // Command from HMI to go to upper position in semiautomatic or manual mode
      CommandDown { ExternalAccessible := 'False'; ExternalVisible := 'False'; ExternalWritable := 'False'} : Bool;   // Command from HMI to go to lower position in semiautomatic or manual mode
      JogUp { ExternalAccessible := 'False'; ExternalVisible := 'False'; ExternalWritable := 'False'} : Bool;   // Command from HMI to Jog upwards
      JogDown { ExternalAccessible := 'False'; ExternalVisible := 'False'; ExternalWritable := 'False'} : Bool;   // Command from HMI to Jog downwards
      ReferenceRun { ExternalAccessible := 'False'; ExternalVisible := 'False'; ExternalWritable := 'False'} : Bool;   // Command from HMI to reference drive
   END_STRUCT;

END_TYPE

TYPE "UDT_VfdConfiguration"
TITLE = UDT_VFD_Configuration
VERSION : 0.1
//User-defined structure oparameters.
   STRUCT
      GearRatio : Real;   // Gear box value X = turns at input to get 1 turn at output
      ReferenceRPM : Real;   // VFD speed max - reference [rpm]
      WheelEndPerimeter : Real;   // Perimeter of wheel at the end of gear [mm]
      VFDRampUpTime : UDInt;   // VFD ramp up time for monitoring starting [ms]
      VFDRampDownTime : UDInt;   // VFD ramp up time for monitoring stopping [ms]
      SpeedSetpointWindow : Int := 5;   // VFD speed setpoint window (tolerance) [mm/s]
      VFDPNDeviceName : String;   // VFD's Profinet device name
      DirectionReversal { ExternalAccessible := 'False'; ExternalVisible := 'False'; ExternalWritable := 'False'} : Bool;   // If true, direction will be swapped
      InterlockFwd { ExternalAccessible := 'False'; ExternalVisible := 'False'; ExternalWritable := 'False'} : Bool;   // False when turning in forward direction is not possible / allowed
      InterlockRvs { ExternalAccessible := 'False'; ExternalVisible := 'False'; ExternalWritable := 'False'} : Bool;   // False when turning in reverse direction is not possible / allowed
      VFDStartupTime : UDInt := 2000;   // Time when the motor should start [ms]
   END_STRUCT;

END_TYPE

TYPE "UDT_VSULiftConfiguration"
TITLE = UDT_VSUConfig
VERSION : 0.1
//User-defined structure of VSU parameters.
   STRUCT
      PEC_GapBeginOnDelay { ExternalAccessible := 'False'; ExternalVisible := 'False'; ExternalWritable := 'False'} : UDInt;   // Photo eye gap begin check time on delay [ms]
      PEC_GapBeginOffDelay { ExternalAccessible := 'False'; ExternalVisible := 'False'; ExternalWritable := 'False'} : UDInt;   // Photo eye  gap begin  check time off delay [ms]
      PEC_GapEndOnDelay { ExternalAccessible := 'False'; ExternalVisible := 'False'; ExternalWritable := 'False'} : UDInt;   // Photo eye gap end check time on delay [ms]
      PEC_GapEndOffDelay { ExternalAccessible := 'False'; ExternalVisible := 'False'; ExternalWritable := 'False'} : UDInt;   // Photo eye  gap end check time off delay [ms]
      JogNoHornTime { ExternalAccessible := 'False'; ExternalVisible := 'False'; ExternalWritable := 'False'} : UDInt := 1000;   // Time within jog buttons can be pressed without new startup indication
      SwitchingTime { ExternalAccessible := 'False'; ExternalVisible := 'False'; ExternalWritable := 'False'} : UInt := 950;   // Time it takes to go from one position to the next [ms]
      DefaultPosition { ExternalAccessible := 'False'; ExternalVisible := 'False'; ExternalWritable := 'False'} : Int := 2;   // Default position number (2= up or 1= down) , If left 0 the block will go to 1
   END_STRUCT;

END_TYPE

TYPE "UDT_ValveConfiguration"
VERSION : 0.1
   STRUCT
      ControlMode : Int := 1;   // 1 = Hold ix_open to keep qx_open active, 2 = detects rising edge on ix_Open to Open, ix_Close to Close
      ValveType : Int := 1;   // 1 = SEV, 2 = DEV
      CloseFeedBackExist { ExternalAccessible := 'False'; ExternalVisible := 'False'; ExternalWritable := 'False'} : Bool;   // Valve has a feed back that signals when fully cLosed
      OpenFeedBackExist { ExternalAccessible := 'False'; ExternalVisible := 'False'; ExternalWritable := 'False'} : Bool;   // Valve has a feed back that signals when fully Open
      OpenTime : Int;   // estimated open time, will trigger FTO if open feedback exist and not detected
      CloseTime : Int;   // estimated close time, will trigger FTC if close feedback exist and not detected
   END_STRUCT;

END_TYPE

TYPE "UDT_UnknownGIN"
TITLE = UDT_UnknownGIN
VERSION : 0.1
//User-defined structure of unknown GIN range.
   STRUCT
      Start : Int := 1;   // Unknown GIN range start value
      End : Int := 199;   // Unknown GIN range end value
      GIN : Int := 0;   // Las generated unknown GIN
   END_STRUCT;

END_TYPE

TYPE "UDT_WSLStatistics"
VERSION : 0.1
   STRUCT
      "010" { ExternalAccessible := 'False'; ExternalVisible := 'False'; ExternalWritable := 'False'} : Struct
         Conveyor { ExternalAccessible := 'False'; ExternalVisible := 'False'; ExternalWritable := 'False'; S7_SetPoint := 'False'} : "UDT_ConveyorStatistics";
         PEC_EoS { ExternalAccessible := 'False'; ExternalVisible := 'False'; ExternalWritable := 'False'} : "UDT_PECStatistics";
         MCO_M01 { ExternalAccessible := 'False'; ExternalVisible := 'False'; ExternalWritable := 'False'; S7_SetPoint := 'False'} : "UDT_VfdStatistics";
      END_STRUCT;
      "020" { ExternalAccessible := 'False'; ExternalVisible := 'False'; ExternalWritable := 'False'} : Struct
         Conveyor { ExternalAccessible := 'False'; ExternalVisible := 'False'; ExternalWritable := 'False'; S7_SetPoint := 'False'} : "UDT_ConveyorStatistics";
         PEC_EoS { ExternalAccessible := 'False'; ExternalVisible := 'False'; ExternalWritable := 'False'} : "UDT_PECStatistics";
         MCO_M01 { ExternalAccessible := 'False'; ExternalVisible := 'False'; ExternalWritable := 'False'; S7_SetPoint := 'False'} : "UDT_VfdStatistics";
      END_STRUCT;
      "030" { ExternalAccessible := 'False'; ExternalVisible := 'False'; ExternalWritable := 'False'} : Struct
         Conveyor { ExternalAccessible := 'False'; ExternalVisible := 'False'; ExternalWritable := 'False'; S7_SetPoint := 'False'} : "UDT_ConveyorStatistics";
         MCO_M01 { ExternalAccessible := 'False'; ExternalVisible := 'False'; ExternalWritable := 'False'; S7_SetPoint := 'False'} : "UDT_VfdStatistics";
      END_STRUCT;
      "040" { ExternalAccessible := 'False'; ExternalVisible := 'False'; ExternalWritable := 'False'} : Struct
         Conveyor { ExternalAccessible := 'False'; ExternalVisible := 'False'; ExternalWritable := 'False'; S7_SetPoint := 'False'} : "UDT_ConveyorStatistics";
         PEC_EoS { ExternalAccessible := 'False'; ExternalVisible := 'False'; ExternalWritable := 'False'} : "UDT_PECStatistics";
         MCO_M01 { ExternalAccessible := 'False'; ExternalVisible := 'False'; ExternalWritable := 'False'; S7_SetPoint := 'False'} : "UDT_VfdStatistics";
      END_STRUCT;
      "050" { ExternalAccessible := 'False'; ExternalVisible := 'False'; ExternalWritable := 'False'} : Struct
         Conveyor { ExternalAccessible := 'False'; ExternalVisible := 'False'; ExternalWritable := 'False'; S7_SetPoint := 'False'} : "UDT_ConveyorStatistics";
         PEC_EoS { ExternalAccessible := 'False'; ExternalVisible := 'False'; ExternalWritable := 'False'} : "UDT_PECStatistics";
         MCO_M01 { ExternalAccessible := 'False'; ExternalVisible := 'False'; ExternalWritable := 'False'; S7_SetPoint := 'False'} : "UDT_VfdStatistics";
      END_STRUCT;
      "060" { ExternalAccessible := 'False'; ExternalVisible := 'False'; ExternalWritable := 'False'} : Struct
         Conveyor { ExternalAccessible := 'False'; ExternalVisible := 'False'; ExternalWritable := 'False'; S7_SetPoint := 'False'} : "UDT_ConveyorStatistics";
         PEC_EoS { ExternalAccessible := 'False'; ExternalVisible := 'False'; ExternalWritable := 'False'} : "UDT_PECStatistics";
         MCO_M01 { ExternalAccessible := 'False'; ExternalVisible := 'False'; ExternalWritable := 'False'; S7_SetPoint := 'False'} : "UDT_VfdStatistics";
      END_STRUCT;
      "070" { ExternalAccessible := 'False'; ExternalVisible := 'False'; ExternalWritable := 'False'} : Struct
         Conveyor { ExternalAccessible := 'False'; ExternalVisible := 'False'; ExternalWritable := 'False'; S7_SetPoint := 'False'} : "UDT_ConveyorStatistics";
         PEC_EoS { ExternalAccessible := 'False'; ExternalVisible := 'False'; ExternalWritable := 'False'} : "UDT_PECStatistics";
         MCO_M01 { ExternalAccessible := 'False'; ExternalVisible := 'False'; ExternalWritable := 'False'; S7_SetPoint := 'False'} : "UDT_VfdStatistics";
      END_STRUCT;
      "080" { ExternalAccessible := 'False'; ExternalVisible := 'False'; ExternalWritable := 'False'} : Struct
         Conveyor { ExternalAccessible := 'False'; ExternalVisible := 'False'; ExternalWritable := 'False'; S7_SetPoint := 'False'} : "UDT_ConveyorStatistics";
         PEC_EoS { ExternalAccessible := 'False'; ExternalVisible := 'False'; ExternalWritable := 'False'} : "UDT_PECStatistics";
         MCO_M01 { ExternalAccessible := 'False'; ExternalVisible := 'False'; ExternalWritable := 'False'; S7_SetPoint := 'False'} : "UDT_VfdStatistics";
      END_STRUCT;
      "090" { ExternalAccessible := 'False'; ExternalVisible := 'False'; ExternalWritable := 'False'} : Struct
         Conveyor { ExternalAccessible := 'False'; ExternalVisible := 'False'; ExternalWritable := 'False'; S7_SetPoint := 'False'} : "UDT_ConveyorStatistics";
         MCO_M01 { ExternalAccessible := 'False'; ExternalVisible := 'False'; ExternalWritable := 'False'; S7_SetPoint := 'False'} : "UDT_VfdStatistics";
      END_STRUCT;
      "100" { ExternalAccessible := 'False'; ExternalVisible := 'False'; ExternalWritable := 'False'} : Struct
         Conveyor { ExternalAccessible := 'False'; ExternalVisible := 'False'; ExternalWritable := 'False'; S7_SetPoint := 'False'} : "UDT_ConveyorStatistics";
         PEC_EoS { ExternalAccessible := 'False'; ExternalVisible := 'False'; ExternalWritable := 'False'} : "UDT_PECStatistics";
         MCO_M01 { ExternalAccessible := 'False'; ExternalVisible := 'False'; ExternalWritable := 'False'; S7_SetPoint := 'False'} : "UDT_VfdStatistics";
      END_STRUCT;
      "110" { ExternalAccessible := 'False'; ExternalVisible := 'False'; ExternalWritable := 'False'} : Struct
         Conveyor { ExternalAccessible := 'False'; ExternalVisible := 'False'; ExternalWritable := 'False'; S7_SetPoint := 'False'} : "UDT_ConveyorStatistics";
         PEC_EoS { ExternalAccessible := 'False'; ExternalVisible := 'False'; ExternalWritable := 'False'} : "UDT_PECStatistics";
         MCO_M01 { ExternalAccessible := 'False'; ExternalVisible := 'False'; ExternalWritable := 'False'; S7_SetPoint := 'False'} : "UDT_VfdStatistics";
      END_STRUCT;
      "120" { ExternalAccessible := 'False'; ExternalVisible := 'False'; ExternalWritable := 'False'} : Struct
         Conveyor { ExternalAccessible := 'False'; ExternalVisible := 'False'; ExternalWritable := 'False'; S7_SetPoint := 'False'} : "UDT_ConveyorStatistics";
         MCO_M01 { ExternalAccessible := 'False'; ExternalVisible := 'False'; ExternalWritable := 'False'; S7_SetPoint := 'False'} : "UDT_VfdStatistics";
      END_STRUCT;
      "121" { ExternalAccessible := 'False'; ExternalVisible := 'False'; ExternalWritable := 'False'} : Struct
         RightAngledTransfer { ExternalAccessible := 'False'; ExternalVisible := 'False'; ExternalWritable := 'False'; S7_SetPoint := 'False'} : "UDT_RATStatistics";
         PEC_EoS { ExternalAccessible := 'False'; ExternalVisible := 'False'; ExternalWritable := 'False'; S7_SetPoint := 'False'} : "UDT_PECStatistics";
         MCO_M01 { ExternalAccessible := 'False'; ExternalVisible := 'False'; ExternalWritable := 'False'; S7_SetPoint := 'False'} : "UDT_VfdStatistics";
      END_STRUCT;
      "210" { ExternalAccessible := 'False'; ExternalVisible := 'False'; ExternalWritable := 'False'} : Struct
         Conveyor { ExternalAccessible := 'False'; ExternalVisible := 'False'; ExternalWritable := 'False'; S7_SetPoint := 'False'} : "UDT_ConveyorStatistics";
         PEC_EoS { ExternalAccessible := 'False'; ExternalVisible := 'False'; ExternalWritable := 'False'} : "UDT_PECStatistics";
         MCO_M01 { ExternalAccessible := 'False'; ExternalVisible := 'False'; ExternalWritable := 'False'; S7_SetPoint := 'False'} : "UDT_VfdStatistics";
      END_STRUCT;
      "220" { ExternalAccessible := 'False'; ExternalVisible := 'False'; ExternalWritable := 'False'} : Struct
         Conveyor { ExternalAccessible := 'False'; ExternalVisible := 'False'; ExternalWritable := 'False'; S7_SetPoint := 'False'} : "UDT_ConveyorStatistics";
         MCO_M01 { ExternalAccessible := 'False'; ExternalVisible := 'False'; ExternalWritable := 'False'; S7_SetPoint := 'False'} : "UDT_VfdStatistics";
      END_STRUCT;
      "221" { ExternalAccessible := 'False'; ExternalVisible := 'False'; ExternalWritable := 'False'} : Struct
         RightAngledTransfer { ExternalAccessible := 'False'; ExternalVisible := 'False'; ExternalWritable := 'False'; S7_SetPoint := 'False'} : "UDT_RATStatistics";
         PEC_EoS { ExternalAccessible := 'False'; ExternalVisible := 'False'; ExternalWritable := 'False'; S7_SetPoint := 'False'} : "UDT_PECStatistics";
         MCO_M01 { ExternalAccessible := 'False'; ExternalVisible := 'False'; ExternalWritable := 'False'; S7_SetPoint := 'False'} : "UDT_VfdStatistics";
      END_STRUCT;
      "230" { ExternalAccessible := 'False'; ExternalVisible := 'False'; ExternalWritable := 'False'} : Struct
         Conveyor { ExternalAccessible := 'False'; ExternalVisible := 'False'; ExternalWritable := 'False'; S7_SetPoint := 'False'} : "UDT_ConveyorStatistics";
         MCO_M01 { ExternalAccessible := 'False'; ExternalVisible := 'False'; ExternalWritable := 'False'; S7_SetPoint := 'False'} : "UDT_VfdStatistics";
      END_STRUCT;
      "240" { ExternalAccessible := 'False'; ExternalVisible := 'False'; ExternalWritable := 'False'} : Struct
         Conveyor { ExternalAccessible := 'False'; ExternalVisible := 'False'; ExternalWritable := 'False'; S7_SetPoint := 'False'} : "UDT_ConveyorStatistics";
         PEC_EoS { ExternalAccessible := 'False'; ExternalVisible := 'False'; ExternalWritable := 'False'} : "UDT_PECStatistics";
         MCO_M01 { ExternalAccessible := 'False'; ExternalVisible := 'False'; ExternalWritable := 'False'; S7_SetPoint := 'False'} : "UDT_VfdStatistics";
      END_STRUCT;
      "250" { ExternalAccessible := 'False'; ExternalVisible := 'False'; ExternalWritable := 'False'} : Struct
         Conveyor { ExternalAccessible := 'False'; ExternalVisible := 'False'; ExternalWritable := 'False'; S7_SetPoint := 'False'} : "UDT_ConveyorStatistics";
         PEC_EoS { ExternalAccessible := 'False'; ExternalVisible := 'False'; ExternalWritable := 'False'} : "UDT_PECStatistics";
         MCO_M01 { ExternalAccessible := 'False'; ExternalVisible := 'False'; ExternalWritable := 'False'; S7_SetPoint := 'False'} : "UDT_VfdStatistics";
      END_STRUCT;
      "260" { ExternalAccessible := 'False'; ExternalVisible := 'False'; ExternalWritable := 'False'} : Struct
         Conveyor { ExternalAccessible := 'False'; ExternalVisible := 'False'; ExternalWritable := 'False'; S7_SetPoint := 'False'} : "UDT_ConveyorStatistics";
         PEC_EoS { ExternalAccessible := 'False'; ExternalVisible := 'False'; ExternalWritable := 'False'} : "UDT_PECStatistics";
         MCO_M01 { ExternalAccessible := 'False'; ExternalVisible := 'False'; ExternalWritable := 'False'; S7_SetPoint := 'False'} : "UDT_VfdStatistics";
      END_STRUCT;
      "270" { ExternalAccessible := 'False'; ExternalVisible := 'False'; ExternalWritable := 'False'} : Struct
         Conveyor { ExternalAccessible := 'False'; ExternalVisible := 'False'; ExternalWritable := 'False'; S7_SetPoint := 'False'} : "UDT_ConveyorStatistics";
         MCO_M01 { ExternalAccessible := 'False'; ExternalVisible := 'False'; ExternalWritable := 'False'; S7_SetPoint := 'False'} : "UDT_VfdStatistics";
      END_STRUCT;
      "280" { ExternalAccessible := 'False'; ExternalVisible := 'False'; ExternalWritable := 'False'} : Struct
         Conveyor { ExternalAccessible := 'False'; ExternalVisible := 'False'; ExternalWritable := 'False'; S7_SetPoint := 'False'} : "UDT_ConveyorStatistics";
         PEC_EoS { ExternalAccessible := 'False'; ExternalVisible := 'False'; ExternalWritable := 'False'} : "UDT_PECStatistics";
         MCO_M01 { ExternalAccessible := 'False'; ExternalVisible := 'False'; ExternalWritable := 'False'; S7_SetPoint := 'False'} : "UDT_VfdStatistics";
      END_STRUCT;
      "290" { ExternalAccessible := 'False'; ExternalVisible := 'False'; ExternalWritable := 'False'} : Struct
         Conveyor { ExternalAccessible := 'False'; ExternalVisible := 'False'; ExternalWritable := 'False'; S7_SetPoint := 'False'} : "UDT_ConveyorStatistics";
         MCO_M01 { ExternalAccessible := 'False'; ExternalVisible := 'False'; ExternalWritable := 'False'; S7_SetPoint := 'False'} : "UDT_VfdStatistics";
      END_STRUCT;
      "291" { ExternalAccessible := 'False'; ExternalVisible := 'False'; ExternalWritable := 'False'} : Struct
         RightAngledTransfer { ExternalAccessible := 'False'; ExternalVisible := 'False'; ExternalWritable := 'False'; S7_SetPoint := 'False'} : "UDT_RATStatistics";
         PEC_EoS { ExternalAccessible := 'False'; ExternalVisible := 'False'; ExternalWritable := 'False'; S7_SetPoint := 'False'} : "UDT_PECStatistics";
         MCO_M01 { ExternalAccessible := 'False'; ExternalVisible := 'False'; ExternalWritable := 'False'; S7_SetPoint := 'False'} : "UDT_VfdStatistics";
      END_STRUCT;
      "300" { ExternalAccessible := 'False'; ExternalVisible := 'False'; ExternalWritable := 'False'} : Struct
         Conveyor { ExternalAccessible := 'False'; ExternalVisible := 'False'; ExternalWritable := 'False'; S7_SetPoint := 'False'} : "UDT_ConveyorStatistics";
         PEC_EoS { ExternalAccessible := 'False'; ExternalVisible := 'False'; ExternalWritable := 'False'} : "UDT_PECStatistics";
         MCO_M01 { ExternalAccessible := 'False'; ExternalVisible := 'False'; ExternalWritable := 'False'; S7_SetPoint := 'False'} : "UDT_VfdStatistics";
      END_STRUCT;
      "410" { ExternalAccessible := 'False'; ExternalVisible := 'False'; ExternalWritable := 'False'} : Struct
         Conveyor { ExternalAccessible := 'False'; ExternalVisible := 'False'; ExternalWritable := 'False'; S7_SetPoint := 'False'} : "UDT_ConveyorStatistics";
         PEC_EoS { ExternalAccessible := 'False'; ExternalVisible := 'False'; ExternalWritable := 'False'} : "UDT_PECStatistics";
         MCO_M01 { ExternalAccessible := 'False'; ExternalVisible := 'False'; ExternalWritable := 'False'; S7_SetPoint := 'False'} : "UDT_VfdStatistics";
      END_STRUCT;
      "420" { ExternalAccessible := 'False'; ExternalVisible := 'False'; ExternalWritable := 'False'} : Struct
         Conveyor { ExternalAccessible := 'False'; ExternalVisible := 'False'; ExternalWritable := 'False'; S7_SetPoint := 'False'} : "UDT_ConveyorStatistics";
         MCO_M01 { ExternalAccessible := 'False'; ExternalVisible := 'False'; ExternalWritable := 'False'; S7_SetPoint := 'False'} : "UDT_VfdStatistics";
      END_STRUCT;
      "421" { ExternalAccessible := 'False'; ExternalVisible := 'False'; ExternalWritable := 'False'} : Struct
         RightAngledTransfer { ExternalAccessible := 'False'; ExternalVisible := 'False'; ExternalWritable := 'False'; S7_SetPoint := 'False'} : "UDT_RATStatistics";
         PEC_EoS { ExternalAccessible := 'False'; ExternalVisible := 'False'; ExternalWritable := 'False'; S7_SetPoint := 'False'} : "UDT_PECStatistics";
         MCO_M01 { ExternalAccessible := 'False'; ExternalVisible := 'False'; ExternalWritable := 'False'; S7_SetPoint := 'False'} : "UDT_VfdStatistics";
      END_STRUCT;
      "430" { ExternalAccessible := 'False'; ExternalVisible := 'False'; ExternalWritable := 'False'} : Struct
         Conveyor { ExternalAccessible := 'False'; ExternalVisible := 'False'; ExternalWritable := 'False'; S7_SetPoint := 'False'} : "UDT_ConveyorStatistics";
         MCO_M01 { ExternalAccessible := 'False'; ExternalVisible := 'False'; ExternalWritable := 'False'; S7_SetPoint := 'False'} : "UDT_VfdStatistics";
      END_STRUCT;
      "440" { ExternalAccessible := 'False'; ExternalVisible := 'False'; ExternalWritable := 'False'} : Struct
         Conveyor { ExternalAccessible := 'False'; ExternalVisible := 'False'; ExternalWritable := 'False'; S7_SetPoint := 'False'} : "UDT_ConveyorStatistics";
         PEC_EoS { ExternalAccessible := 'False'; ExternalVisible := 'False'; ExternalWritable := 'False'} : "UDT_PECStatistics";
         MCO_M01 { ExternalAccessible := 'False'; ExternalVisible := 'False'; ExternalWritable := 'False'; S7_SetPoint := 'False'} : "UDT_VfdStatistics";
      END_STRUCT;
      "450" { ExternalAccessible := 'False'; ExternalVisible := 'False'; ExternalWritable := 'False'} : Struct
         Conveyor { ExternalAccessible := 'False'; ExternalVisible := 'False'; ExternalWritable := 'False'; S7_SetPoint := 'False'} : "UDT_ConveyorStatistics";
         PEC_EoS { ExternalAccessible := 'False'; ExternalVisible := 'False'; ExternalWritable := 'False'} : "UDT_PECStatistics";
         MCO_M01 { ExternalAccessible := 'False'; ExternalVisible := 'False'; ExternalWritable := 'False'; S7_SetPoint := 'False'} : "UDT_VfdStatistics";
      END_STRUCT;
      "460" { ExternalAccessible := 'False'; ExternalVisible := 'False'; ExternalWritable := 'False'} : Struct
         Conveyor { ExternalAccessible := 'False'; ExternalVisible := 'False'; ExternalWritable := 'False'; S7_SetPoint := 'False'} : "UDT_ConveyorStatistics";
         PEC_EoS { ExternalAccessible := 'False'; ExternalVisible := 'False'; ExternalWritable := 'False'} : "UDT_PECStatistics";
         MCO_M01 { ExternalAccessible := 'False'; ExternalVisible := 'False'; ExternalWritable := 'False'; S7_SetPoint := 'False'} : "UDT_VfdStatistics";
      END_STRUCT;
      "470" { ExternalAccessible := 'False'; ExternalVisible := 'False'; ExternalWritable := 'False'} : Struct
         Conveyor { ExternalAccessible := 'False'; ExternalVisible := 'False'; ExternalWritable := 'False'; S7_SetPoint := 'False'} : "UDT_ConveyorStatistics";
         MCO_M01 { ExternalAccessible := 'False'; ExternalVisible := 'False'; ExternalWritable := 'False'; S7_SetPoint := 'False'} : "UDT_VfdStatistics";
      END_STRUCT;
      "480" { ExternalAccessible := 'False'; ExternalVisible := 'False'; ExternalWritable := 'False'} : Struct
         Conveyor { ExternalAccessible := 'False'; ExternalVisible := 'False'; ExternalWritable := 'False'; S7_SetPoint := 'False'} : "UDT_ConveyorStatistics";
         PEC_EoS { ExternalAccessible := 'False'; ExternalVisible := 'False'; ExternalWritable := 'False'} : "UDT_PECStatistics";
         MCO_M01 { ExternalAccessible := 'False'; ExternalVisible := 'False'; ExternalWritable := 'False'; S7_SetPoint := 'False'} : "UDT_VfdStatistics";
      END_STRUCT;
      "490" { ExternalAccessible := 'False'; ExternalVisible := 'False'; ExternalWritable := 'False'} : Struct
         Conveyor { ExternalAccessible := 'False'; ExternalVisible := 'False'; ExternalWritable := 'False'; S7_SetPoint := 'False'} : "UDT_ConveyorStatistics";
         MCO_M01 { ExternalAccessible := 'False'; ExternalVisible := 'False'; ExternalWritable := 'False'; S7_SetPoint := 'False'} : "UDT_VfdStatistics";
      END_STRUCT;
      "491" { ExternalAccessible := 'False'; ExternalVisible := 'False'; ExternalWritable := 'False'} : Struct
         RightAngledTransfer { ExternalAccessible := 'False'; ExternalVisible := 'False'; ExternalWritable := 'False'; S7_SetPoint := 'False'} : "UDT_RATStatistics";
         PEC_EoS { ExternalAccessible := 'False'; ExternalVisible := 'False'; ExternalWritable := 'False'; S7_SetPoint := 'False'} : "UDT_PECStatistics";
         MCO_M01 { ExternalAccessible := 'False'; ExternalVisible := 'False'; ExternalWritable := 'False'; S7_SetPoint := 'False'} : "UDT_VfdStatistics";
      END_STRUCT;
      "500" { ExternalAccessible := 'False'; ExternalVisible := 'False'; ExternalWritable := 'False'} : Struct
         Conveyor { ExternalAccessible := 'False'; ExternalVisible := 'False'; ExternalWritable := 'False'; S7_SetPoint := 'False'} : "UDT_ConveyorStatistics";
         PEC_EoS { ExternalAccessible := 'False'; ExternalVisible := 'False'; ExternalWritable := 'False'} : "UDT_PECStatistics";
         MCO_M01 { ExternalAccessible := 'False'; ExternalVisible := 'False'; ExternalWritable := 'False'; S7_SetPoint := 'False'} : "UDT_VfdStatistics";
      END_STRUCT;
      "610" { ExternalAccessible := 'False'; ExternalVisible := 'False'; ExternalWritable := 'False'} : Struct
         Conveyor { ExternalAccessible := 'False'; ExternalVisible := 'False'; ExternalWritable := 'False'; S7_SetPoint := 'False'} : "UDT_ConveyorStatistics";
         MCO_M01 { ExternalAccessible := 'False'; ExternalVisible := 'False'; ExternalWritable := 'False'; S7_SetPoint := 'False'} : "UDT_VfdStatistics";
      END_STRUCT;
      "611" { ExternalAccessible := 'False'; ExternalVisible := 'False'; ExternalWritable := 'False'} : Struct
         RightAngledTransfer { ExternalAccessible := 'False'; ExternalVisible := 'False'; ExternalWritable := 'False'; S7_SetPoint := 'False'} : "UDT_RATStatistics";
         PEC_EoS { ExternalAccessible := 'False'; ExternalVisible := 'False'; ExternalWritable := 'False'; S7_SetPoint := 'False'} : "UDT_PECStatistics";
         MCO_M01 { ExternalAccessible := 'False'; ExternalVisible := 'False'; ExternalWritable := 'False'; S7_SetPoint := 'False'} : "UDT_VfdStatistics";
      END_STRUCT;
      "620" { ExternalAccessible := 'False'; ExternalVisible := 'False'; ExternalWritable := 'False'} : Struct
         Conveyor { ExternalAccessible := 'False'; ExternalVisible := 'False'; ExternalWritable := 'False'; S7_SetPoint := 'False'} : "UDT_ConveyorStatistics";
         MCO_M01 { ExternalAccessible := 'False'; ExternalVisible := 'False'; ExternalWritable := 'False'; S7_SetPoint := 'False'} : "UDT_VfdStatistics";
      END_STRUCT;
      "630" { ExternalAccessible := 'False'; ExternalVisible := 'False'; ExternalWritable := 'False'} : Struct
         Conveyor { ExternalAccessible := 'False'; ExternalVisible := 'False'; ExternalWritable := 'False'; S7_SetPoint := 'False'} : "UDT_ConveyorStatistics";
         MCO_M01 { ExternalAccessible := 'False'; ExternalVisible := 'False'; ExternalWritable := 'False'; S7_SetPoint := 'False'} : "UDT_VfdStatistics";
      END_STRUCT;
      "640" { ExternalAccessible := 'False'; ExternalVisible := 'False'; ExternalWritable := 'False'} : Struct
         Conveyor { ExternalAccessible := 'False'; ExternalVisible := 'False'; ExternalWritable := 'False'; S7_SetPoint := 'False'} : "UDT_ConveyorStatistics";
         PEC_EoS { ExternalAccessible := 'False'; ExternalVisible := 'False'; ExternalWritable := 'False'} : "UDT_PECStatistics";
         MCO_M01 { ExternalAccessible := 'False'; ExternalVisible := 'False'; ExternalWritable := 'False'; S7_SetPoint := 'False'} : "UDT_VfdStatistics";
      END_STRUCT;
   END_STRUCT;

END_TYPE

TYPE "UDT_WSLHmiCommands"
VERSION : 0.1
   STRUCT
      "010" : Struct
         Conveyor { S7_SetPoint := 'False'} : "UDT_ConveyorCommand";
      END_STRUCT;
      "020" : Struct
         Conveyor { S7_SetPoint := 'False'} : "UDT_ConveyorCommand";
      END_STRUCT;
      "030" : Struct
         Conveyor { S7_SetPoint := 'False'} : "UDT_ConveyorCommand";
      END_STRUCT;
      "040" : Struct
         Conveyor { S7_SetPoint := 'False'} : "UDT_ConveyorCommand";
      END_STRUCT;
      "050" : Struct
         Conveyor { S7_SetPoint := 'False'} : "UDT_ConveyorCommand";
      END_STRUCT;
      "060" : Struct
         Conveyor { S7_SetPoint := 'False'} : "UDT_ConveyorCommand";
      END_STRUCT;
      "070" : Struct
         Conveyor { S7_SetPoint := 'False'} : "UDT_ConveyorCommand";
      END_STRUCT;
      "080" : Struct
         Conveyor { S7_SetPoint := 'False'} : "UDT_ConveyorCommand";
      END_STRUCT;
      "090" : Struct
         Conveyor { S7_SetPoint := 'False'} : "UDT_ConveyorCommand";
      END_STRUCT;
      "100" : Struct
         Conveyor { S7_SetPoint := 'False'} : "UDT_ConveyorCommand";
      END_STRUCT;
      "110" : Struct
         Conveyor { S7_SetPoint := 'False'} : "UDT_ConveyorCommand";
      END_STRUCT;
      "120" : Struct
         Conveyor { S7_SetPoint := 'False'} : "UDT_ConveyorCommand";
      END_STRUCT;
      "121" : Struct
         RightAngledTransfer { S7_SetPoint := 'False'} : "UDT_RATCommand";
      END_STRUCT;
      "210" : Struct
         Conveyor { S7_SetPoint := 'False'} : "UDT_ConveyorCommand";
      END_STRUCT;
      "220" : Struct
         Conveyor { S7_SetPoint := 'False'} : "UDT_ConveyorCommand";
      END_STRUCT;
      "221" : Struct
         RightAngledTransfer { S7_SetPoint := 'False'} : "UDT_RATCommand";
      END_STRUCT;
      "230" : Struct
         Conveyor { S7_SetPoint := 'False'} : "UDT_ConveyorCommand";
      END_STRUCT;
      "240" : Struct
         Conveyor { S7_SetPoint := 'False'} : "UDT_ConveyorCommand";
      END_STRUCT;
      "250" : Struct
         Conveyor { S7_SetPoint := 'False'} : "UDT_ConveyorCommand";
      END_STRUCT;
      "260" : Struct
         Conveyor { S7_SetPoint := 'False'} : "UDT_ConveyorCommand";
      END_STRUCT;
      "270" : Struct
         Conveyor { S7_SetPoint := 'False'} : "UDT_ConveyorCommand";
      END_STRUCT;
      "280" : Struct
         Conveyor { S7_SetPoint := 'False'} : "UDT_ConveyorCommand";
      END_STRUCT;
      "290" : Struct
         Conveyor { S7_SetPoint := 'False'} : "UDT_ConveyorCommand";
      END_STRUCT;
      "291" : Struct
         RightAngledTransfer { S7_SetPoint := 'False'} : "UDT_RATCommand";
      END_STRUCT;
      "300" : Struct
         Conveyor { S7_SetPoint := 'False'} : "UDT_ConveyorCommand";
      END_STRUCT;
      "410" : Struct
         Conveyor { S7_SetPoint := 'False'} : "UDT_ConveyorCommand";
      END_STRUCT;
      "420" : Struct
         Conveyor { S7_SetPoint := 'False'} : "UDT_ConveyorCommand";
      END_STRUCT;
      "421" : Struct
         RightAngledTransfer { S7_SetPoint := 'False'} : "UDT_RATCommand";
      END_STRUCT;
      "430" : Struct
         Conveyor { S7_SetPoint := 'False'} : "UDT_ConveyorCommand";
      END_STRUCT;
      "440" : Struct
         Conveyor { S7_SetPoint := 'False'} : "UDT_ConveyorCommand";
      END_STRUCT;
      "450" : Struct
         Conveyor { S7_SetPoint := 'False'} : "UDT_ConveyorCommand";
      END_STRUCT;
      "460" : Struct
         Conveyor { S7_SetPoint := 'False'} : "UDT_ConveyorCommand";
      END_STRUCT;
      "470" : Struct
         Conveyor { S7_SetPoint := 'False'} : "UDT_ConveyorCommand";
      END_STRUCT;
      "480" : Struct
         Conveyor { S7_SetPoint := 'False'} : "UDT_ConveyorCommand";
      END_STRUCT;
      "490" : Struct
         Conveyor { S7_SetPoint := 'False'} : "UDT_ConveyorCommand";
      END_STRUCT;
      "491" : Struct
         RAT { S7_SetPoint := 'False'} : "UDT_RATCommand";
      END_STRUCT;
      "500" : Struct
         Conveyor { S7_SetPoint := 'False'} : "UDT_ConveyorCommand";
      END_STRUCT;
      "610" : Struct
         Conveyor { S7_SetPoint := 'False'} : "UDT_ConveyorCommand";
      END_STRUCT;
      "611" : Struct
         RightAngledTransfer { S7_SetPoint := 'False'} : "UDT_RATCommand";
      END_STRUCT;
      "620" : Struct
         Conveyor { S7_SetPoint := 'False'} : "UDT_ConveyorCommand";
      END_STRUCT;
      "630" : Struct
         Conveyor { S7_SetPoint := 'False'} : "UDT_ConveyorCommand";
      END_STRUCT;
      "640" : Struct
         Conveyor { S7_SetPoint := 'False'} : "UDT_ConveyorCommand";
      END_STRUCT;
   END_STRUCT;

END_TYPE

TYPE "UDT_WSLConfiguration"
VERSION : 0.1
   STRUCT
      GlobalConfig { ExternalAccessible := 'False'; ExternalVisible := 'False'; ExternalWritable := 'False'} : Struct
         LeftStationExists { ExternalAccessible := 'False'; ExternalVisible := 'False'; ExternalWritable := 'False'} : Bool := TRUE;
         RightStationExists { ExternalAccessible := 'False'; ExternalVisible := 'False'; ExternalWritable := 'False'} : Bool := TRUE;
      END_STRUCT;
      "010" { ExternalAccessible := 'False'; ExternalVisible := 'False'; ExternalWritable := 'False'} : Struct
         Conveyor { ExternalAccessible := 'False'; ExternalVisible := 'False'; ExternalWritable := 'False'; S7_SetPoint := 'False'} : "UDT_ConveyorConfiguration";
         PEC_EoS { ExternalAccessible := 'False'; ExternalVisible := 'False'; ExternalWritable := 'False'} : "UDT_PECConfiguration";
         MCO_M01 { ExternalAccessible := 'False'; ExternalVisible := 'False'; ExternalWritable := 'False'} : "UDT_AixPlcFullControllerConfiguration";
      END_STRUCT;
      "020" { ExternalAccessible := 'False'; ExternalVisible := 'False'; ExternalWritable := 'False'} : Struct
         Conveyor { ExternalAccessible := 'False'; ExternalVisible := 'False'; ExternalWritable := 'False'; S7_SetPoint := 'False'} : "UDT_ConveyorConfiguration";
         PEC_EoS { ExternalAccessible := 'False'; ExternalVisible := 'False'; ExternalWritable := 'False'} : "UDT_PECConfiguration";
         MCO_M01 { ExternalAccessible := 'False'; ExternalVisible := 'False'; ExternalWritable := 'False'} : "UDT_AixPlcFullControllerConfiguration";
      END_STRUCT;
      "030" { ExternalAccessible := 'False'; ExternalVisible := 'False'; ExternalWritable := 'False'} : Struct
         Conveyor { ExternalAccessible := 'False'; ExternalVisible := 'False'; ExternalWritable := 'False'; S7_SetPoint := 'False'} : "UDT_ConveyorConfiguration";
         MCO_M01 { ExternalAccessible := 'False'; ExternalVisible := 'False'; ExternalWritable := 'False'} : "UDT_AixPlcFullControllerConfiguration";
      END_STRUCT;
      "040" { ExternalAccessible := 'False'; ExternalVisible := 'False'; ExternalWritable := 'False'} : Struct
         Conveyor { ExternalAccessible := 'False'; ExternalVisible := 'False'; ExternalWritable := 'False'; S7_SetPoint := 'False'} : "UDT_ConveyorConfiguration";
         PEC_EoS { ExternalAccessible := 'False'; ExternalVisible := 'False'; ExternalWritable := 'False'} : "UDT_PECConfiguration";
         MCO_M01 { ExternalAccessible := 'False'; ExternalVisible := 'False'; ExternalWritable := 'False'} : "UDT_AixPlcFullControllerConfiguration";
      END_STRUCT;
      "050" { ExternalAccessible := 'False'; ExternalVisible := 'False'; ExternalWritable := 'False'} : Struct
         Conveyor { ExternalAccessible := 'False'; ExternalVisible := 'False'; ExternalWritable := 'False'; S7_SetPoint := 'False'} : "UDT_ConveyorConfiguration";
         PEC_EoS { ExternalAccessible := 'False'; ExternalVisible := 'False'; ExternalWritable := 'False'} : "UDT_PECConfiguration";
         MCO_M01 { ExternalAccessible := 'False'; ExternalVisible := 'False'; ExternalWritable := 'False'} : "UDT_AixPlcFullControllerConfiguration";
      END_STRUCT;
      "060" { ExternalAccessible := 'False'; ExternalVisible := 'False'; ExternalWritable := 'False'} : Struct
         Conveyor { ExternalAccessible := 'False'; ExternalVisible := 'False'; ExternalWritable := 'False'; S7_SetPoint := 'False'} : "UDT_ConveyorConfiguration";
         PEC_EoS { ExternalAccessible := 'False'; ExternalVisible := 'False'; ExternalWritable := 'False'} : "UDT_PECConfiguration";
         MCO_M01 { ExternalAccessible := 'False'; ExternalVisible := 'False'; ExternalWritable := 'False'} : "UDT_AixPlcFullControllerConfiguration";
      END_STRUCT;
      "070" { ExternalAccessible := 'False'; ExternalVisible := 'False'; ExternalWritable := 'False'} : Struct
         Conveyor { ExternalAccessible := 'False'; ExternalVisible := 'False'; ExternalWritable := 'False'; S7_SetPoint := 'False'} : "UDT_ConveyorConfiguration";
         PEC_EoS { ExternalAccessible := 'False'; ExternalVisible := 'False'; ExternalWritable := 'False'} : "UDT_PECConfiguration";
         MCO_M01 { ExternalAccessible := 'False'; ExternalVisible := 'False'; ExternalWritable := 'False'} : "UDT_AixPlcFullControllerConfiguration";
      END_STRUCT;
      "080" { ExternalAccessible := 'False'; ExternalVisible := 'False'; ExternalWritable := 'False'} : Struct
         Conveyor { ExternalAccessible := 'False'; ExternalVisible := 'False'; ExternalWritable := 'False'; S7_SetPoint := 'False'} : "UDT_ConveyorConfiguration";
         PEC_EoS { ExternalAccessible := 'False'; ExternalVisible := 'False'; ExternalWritable := 'False'} : "UDT_PECConfiguration";
         MCO_M01 { ExternalAccessible := 'False'; ExternalVisible := 'False'; ExternalWritable := 'False'} : "UDT_AixPlcFullControllerConfiguration";
      END_STRUCT;
      "090" { ExternalAccessible := 'False'; ExternalVisible := 'False'; ExternalWritable := 'False'} : Struct
         Conveyor { ExternalAccessible := 'False'; ExternalVisible := 'False'; ExternalWritable := 'False'; S7_SetPoint := 'False'} : "UDT_ConveyorConfiguration";
         MCO_M01 { ExternalAccessible := 'False'; ExternalVisible := 'False'; ExternalWritable := 'False'} : "UDT_AixPlcFullControllerConfiguration";
      END_STRUCT;
      "100" { ExternalAccessible := 'False'; ExternalVisible := 'False'; ExternalWritable := 'False'} : Struct
         Conveyor { ExternalAccessible := 'False'; ExternalVisible := 'False'; ExternalWritable := 'False'; S7_SetPoint := 'False'} : "UDT_ConveyorConfiguration";
         PEC_EoS { ExternalAccessible := 'False'; ExternalVisible := 'False'; ExternalWritable := 'False'} : "UDT_PECConfiguration";
         MCO_M01 { ExternalAccessible := 'False'; ExternalVisible := 'False'; ExternalWritable := 'False'} : "UDT_AixPlcFullControllerConfiguration";
      END_STRUCT;
      "110" { ExternalAccessible := 'False'; ExternalVisible := 'False'; ExternalWritable := 'False'} : Struct
         Conveyor { ExternalAccessible := 'False'; ExternalVisible := 'False'; ExternalWritable := 'False'; S7_SetPoint := 'False'} : "UDT_ConveyorConfiguration";
         PEC_EoS { ExternalAccessible := 'False'; ExternalVisible := 'False'; ExternalWritable := 'False'} : "UDT_PECConfiguration";
         MCO_M01 { ExternalAccessible := 'False'; ExternalVisible := 'False'; ExternalWritable := 'False'} : "UDT_AixPlcFullControllerConfiguration";
      END_STRUCT;
      "120" { ExternalAccessible := 'False'; ExternalVisible := 'False'; ExternalWritable := 'False'} : Struct
         Conveyor { ExternalAccessible := 'False'; ExternalVisible := 'False'; ExternalWritable := 'False'; S7_SetPoint := 'False'} : "UDT_ConveyorConfiguration";
         PEC_EoS { ExternalAccessible := 'False'; ExternalVisible := 'False'; ExternalWritable := 'False'} : "UDT_PECConfiguration";
         MCO_M01 { ExternalAccessible := 'False'; ExternalVisible := 'False'; ExternalWritable := 'False'} : "UDT_AixPlcFullControllerConfiguration";
      END_STRUCT;
      "121" { ExternalAccessible := 'False'; ExternalVisible := 'False'; ExternalWritable := 'False'} : Struct
         Conveyor { ExternalAccessible := 'False'; ExternalVisible := 'False'; ExternalWritable := 'False'; S7_SetPoint := 'False'} : "UDT_ConveyorConfiguration";
         RightAngledTransfer { ExternalAccessible := 'False'; ExternalVisible := 'False'; ExternalWritable := 'False'; S7_SetPoint := 'False'} : "UDT_RATConfiguration";
         MCO_M01 { ExternalAccessible := 'False'; ExternalVisible := 'False'; ExternalWritable := 'False'} : "UDT_AixPlcFullControllerConfiguration";
      END_STRUCT;
      "210" { ExternalAccessible := 'False'; ExternalVisible := 'False'; ExternalWritable := 'False'} : Struct
         Conveyor { ExternalAccessible := 'False'; ExternalVisible := 'False'; ExternalWritable := 'False'; S7_SetPoint := 'False'} : "UDT_ConveyorConfiguration";
         PEC_EoS { ExternalAccessible := 'False'; ExternalVisible := 'False'; ExternalWritable := 'False'} : "UDT_PECConfiguration";
         MCO_M01 { ExternalAccessible := 'False'; ExternalVisible := 'False'; ExternalWritable := 'False'} : "UDT_AixPlcFullControllerConfiguration";
      END_STRUCT;
      "220" { ExternalAccessible := 'False'; ExternalVisible := 'False'; ExternalWritable := 'False'} : Struct
         Conveyor { ExternalAccessible := 'False'; ExternalVisible := 'False'; ExternalWritable := 'False'; S7_SetPoint := 'False'} : "UDT_ConveyorConfiguration";
         PEC_EoS { ExternalAccessible := 'False'; ExternalVisible := 'False'; ExternalWritable := 'False'} : "UDT_PECConfiguration";
         MCO_M01 { ExternalAccessible := 'False'; ExternalVisible := 'False'; ExternalWritable := 'False'} : "UDT_AixPlcFullControllerConfiguration";
      END_STRUCT;
      "221" { ExternalAccessible := 'False'; ExternalVisible := 'False'; ExternalWritable := 'False'} : Struct
         Conveyor { ExternalAccessible := 'False'; ExternalVisible := 'False'; ExternalWritable := 'False'; S7_SetPoint := 'False'} : "UDT_ConveyorConfiguration";
         RightAngledTransfer { ExternalAccessible := 'False'; ExternalVisible := 'False'; ExternalWritable := 'False'; S7_SetPoint := 'False'} : "UDT_RATConfiguration";
         MCO_M01 { ExternalAccessible := 'False'; ExternalVisible := 'False'; ExternalWritable := 'False'} : "UDT_AixPlcFullControllerConfiguration";
      END_STRUCT;
      "230" { ExternalAccessible := 'False'; ExternalVisible := 'False'; ExternalWritable := 'False'} : Struct
         Conveyor { ExternalAccessible := 'False'; ExternalVisible := 'False'; ExternalWritable := 'False'; S7_SetPoint := 'False'} : "UDT_ConveyorConfiguration";
         MCO_M01 { ExternalAccessible := 'False'; ExternalVisible := 'False'; ExternalWritable := 'False'} : "UDT_AixPlcFullControllerConfiguration";
      END_STRUCT;
      "240" { ExternalAccessible := 'False'; ExternalVisible := 'False'; ExternalWritable := 'False'} : Struct
         Conveyor { ExternalAccessible := 'False'; ExternalVisible := 'False'; ExternalWritable := 'False'; S7_SetPoint := 'False'} : "UDT_ConveyorConfiguration";
         PEC_EoS { ExternalAccessible := 'False'; ExternalVisible := 'False'; ExternalWritable := 'False'} : "UDT_PECConfiguration";
         MCO_M01 { ExternalAccessible := 'False'; ExternalVisible := 'False'; ExternalWritable := 'False'} : "UDT_AixPlcFullControllerConfiguration";
      END_STRUCT;
      "250" { ExternalAccessible := 'False'; ExternalVisible := 'False'; ExternalWritable := 'False'} : Struct
         Conveyor { ExternalAccessible := 'False'; ExternalVisible := 'False'; ExternalWritable := 'False'; S7_SetPoint := 'False'} : "UDT_ConveyorConfiguration";
         PEC_EoS { ExternalAccessible := 'False'; ExternalVisible := 'False'; ExternalWritable := 'False'} : "UDT_PECConfiguration";
         MCO_M01 { ExternalAccessible := 'False'; ExternalVisible := 'False'; ExternalWritable := 'False'} : "UDT_AixPlcFullControllerConfiguration";
      END_STRUCT;
      "260" { ExternalAccessible := 'False'; ExternalVisible := 'False'; ExternalWritable := 'False'} : Struct
         Conveyor { ExternalAccessible := 'False'; ExternalVisible := 'False'; ExternalWritable := 'False'; S7_SetPoint := 'False'} : "UDT_ConveyorConfiguration";
         PEC_EoS { ExternalAccessible := 'False'; ExternalVisible := 'False'; ExternalWritable := 'False'} : "UDT_PECConfiguration";
         MCO_M01 { ExternalAccessible := 'False'; ExternalVisible := 'False'; ExternalWritable := 'False'} : "UDT_AixPlcFullControllerConfiguration";
      END_STRUCT;
      "270" { ExternalAccessible := 'False'; ExternalVisible := 'False'; ExternalWritable := 'False'} : Struct
         Conveyor { ExternalAccessible := 'False'; ExternalVisible := 'False'; ExternalWritable := 'False'; S7_SetPoint := 'False'} : "UDT_ConveyorConfiguration";
         MCO_M01 { ExternalAccessible := 'False'; ExternalVisible := 'False'; ExternalWritable := 'False'} : "UDT_AixPlcFullControllerConfiguration";
      END_STRUCT;
      "280" { ExternalAccessible := 'False'; ExternalVisible := 'False'; ExternalWritable := 'False'} : Struct
         Conveyor { ExternalAccessible := 'False'; ExternalVisible := 'False'; ExternalWritable := 'False'; S7_SetPoint := 'False'} : "UDT_ConveyorConfiguration";
         PEC_EoS { ExternalAccessible := 'False'; ExternalVisible := 'False'; ExternalWritable := 'False'} : "UDT_PECConfiguration";
         MCO_M01 { ExternalAccessible := 'False'; ExternalVisible := 'False'; ExternalWritable := 'False'} : "UDT_AixPlcFullControllerConfiguration";
      END_STRUCT;
      "290" { ExternalAccessible := 'False'; ExternalVisible := 'False'; ExternalWritable := 'False'} : Struct
         Conveyor { ExternalAccessible := 'False'; ExternalVisible := 'False'; ExternalWritable := 'False'; S7_SetPoint := 'False'} : "UDT_ConveyorConfiguration";
         PEC_EoS { ExternalAccessible := 'False'; ExternalVisible := 'False'; ExternalWritable := 'False'} : "UDT_PECConfiguration";
         MCO_M01 { ExternalAccessible := 'False'; ExternalVisible := 'False'; ExternalWritable := 'False'} : "UDT_AixPlcFullControllerConfiguration";
      END_STRUCT;
      "291" { ExternalAccessible := 'False'; ExternalVisible := 'False'; ExternalWritable := 'False'} : Struct
         Conveyor { ExternalAccessible := 'False'; ExternalVisible := 'False'; ExternalWritable := 'False'; S7_SetPoint := 'False'} : "UDT_ConveyorConfiguration";
         RightAngledTransfer { ExternalAccessible := 'False'; ExternalVisible := 'False'; ExternalWritable := 'False'; S7_SetPoint := 'False'} : "UDT_RATConfiguration";
         MCO_M01 { ExternalAccessible := 'False'; ExternalVisible := 'False'; ExternalWritable := 'False'} : "UDT_AixPlcFullControllerConfiguration";
      END_STRUCT;
      "300" { ExternalAccessible := 'False'; ExternalVisible := 'False'; ExternalWritable := 'False'} : Struct
         Conveyor { ExternalAccessible := 'False'; ExternalVisible := 'False'; ExternalWritable := 'False'; S7_SetPoint := 'False'} : "UDT_ConveyorConfiguration";
         PEC_EoS { ExternalAccessible := 'False'; ExternalVisible := 'False'; ExternalWritable := 'False'} : "UDT_PECConfiguration";
         MCO_M01 { ExternalAccessible := 'False'; ExternalVisible := 'False'; ExternalWritable := 'False'} : "UDT_AixPlcFullControllerConfiguration";
      END_STRUCT;
      "410" { ExternalAccessible := 'False'; ExternalVisible := 'False'; ExternalWritable := 'False'} : Struct
         Conveyor { ExternalAccessible := 'False'; ExternalVisible := 'False'; ExternalWritable := 'False'; S7_SetPoint := 'False'} : "UDT_ConveyorConfiguration";
         PEC_EoS { ExternalAccessible := 'False'; ExternalVisible := 'False'; ExternalWritable := 'False'} : "UDT_PECConfiguration";
         MCO_M01 { ExternalAccessible := 'False'; ExternalVisible := 'False'; ExternalWritable := 'False'} : "UDT_AixPlcFullControllerConfiguration";
      END_STRUCT;
      "420" { ExternalAccessible := 'False'; ExternalVisible := 'False'; ExternalWritable := 'False'} : Struct
         Conveyor { ExternalAccessible := 'False'; ExternalVisible := 'False'; ExternalWritable := 'False'; S7_SetPoint := 'False'} : "UDT_ConveyorConfiguration";
         PEC_EoS { ExternalAccessible := 'False'; ExternalVisible := 'False'; ExternalWritable := 'False'} : "UDT_PECConfiguration";
         MCO_M01 { ExternalAccessible := 'False'; ExternalVisible := 'False'; ExternalWritable := 'False'} : "UDT_AixPlcFullControllerConfiguration";
      END_STRUCT;
      "421" { ExternalAccessible := 'False'; ExternalVisible := 'False'; ExternalWritable := 'False'} : Struct
         Conveyor { ExternalAccessible := 'False'; ExternalVisible := 'False'; ExternalWritable := 'False'; S7_SetPoint := 'False'} : "UDT_ConveyorConfiguration";
         RightAngledTransfer { ExternalAccessible := 'False'; ExternalVisible := 'False'; ExternalWritable := 'False'; S7_SetPoint := 'False'} : "UDT_RATConfiguration";
         MCO_M01 { ExternalAccessible := 'False'; ExternalVisible := 'False'; ExternalWritable := 'False'} : "UDT_AixPlcFullControllerConfiguration";
      END_STRUCT;
      "430" { ExternalAccessible := 'False'; ExternalVisible := 'False'; ExternalWritable := 'False'} : Struct
         Conveyor { ExternalAccessible := 'False'; ExternalVisible := 'False'; ExternalWritable := 'False'; S7_SetPoint := 'False'} : "UDT_ConveyorConfiguration";
         MCO_M01 { ExternalAccessible := 'False'; ExternalVisible := 'False'; ExternalWritable := 'False'} : "UDT_AixPlcFullControllerConfiguration";
      END_STRUCT;
      "440" { ExternalAccessible := 'False'; ExternalVisible := 'False'; ExternalWritable := 'False'} : Struct
         Conveyor { ExternalAccessible := 'False'; ExternalVisible := 'False'; ExternalWritable := 'False'; S7_SetPoint := 'False'} : "UDT_ConveyorConfiguration";
         PEC_EoS { ExternalAccessible := 'False'; ExternalVisible := 'False'; ExternalWritable := 'False'} : "UDT_PECConfiguration";
         MCO_M01 { ExternalAccessible := 'False'; ExternalVisible := 'False'; ExternalWritable := 'False'} : "UDT_AixPlcFullControllerConfiguration";
      END_STRUCT;
      "450" { ExternalAccessible := 'False'; ExternalVisible := 'False'; ExternalWritable := 'False'} : Struct
         Conveyor { ExternalAccessible := 'False'; ExternalVisible := 'False'; ExternalWritable := 'False'; S7_SetPoint := 'False'} : "UDT_ConveyorConfiguration";
         PEC_EoS { ExternalAccessible := 'False'; ExternalVisible := 'False'; ExternalWritable := 'False'} : "UDT_PECConfiguration";
         MCO_M01 { ExternalAccessible := 'False'; ExternalVisible := 'False'; ExternalWritable := 'False'} : "UDT_AixPlcFullControllerConfiguration";
      END_STRUCT;
      "460" { ExternalAccessible := 'False'; ExternalVisible := 'False'; ExternalWritable := 'False'} : Struct
         Conveyor { ExternalAccessible := 'False'; ExternalVisible := 'False'; ExternalWritable := 'False'; S7_SetPoint := 'False'} : "UDT_ConveyorConfiguration";
         PEC_EoS { ExternalAccessible := 'False'; ExternalVisible := 'False'; ExternalWritable := 'False'} : "UDT_PECConfiguration";
         MCO_M01 { ExternalAccessible := 'False'; ExternalVisible := 'False'; ExternalWritable := 'False'} : "UDT_AixPlcFullControllerConfiguration";
      END_STRUCT;
      "470" { ExternalAccessible := 'False'; ExternalVisible := 'False'; ExternalWritable := 'False'} : Struct
         Conveyor { ExternalAccessible := 'False'; ExternalVisible := 'False'; ExternalWritable := 'False'; S7_SetPoint := 'False'} : "UDT_ConveyorConfiguration";
         MCO_M01 { ExternalAccessible := 'False'; ExternalVisible := 'False'; ExternalWritable := 'False'} : "UDT_AixPlcFullControllerConfiguration";
      END_STRUCT;
      "480" { ExternalAccessible := 'False'; ExternalVisible := 'False'; ExternalWritable := 'False'} : Struct
         Conveyor { ExternalAccessible := 'False'; ExternalVisible := 'False'; ExternalWritable := 'False'; S7_SetPoint := 'False'} : "UDT_ConveyorConfiguration";
         PEC_EoS { ExternalAccessible := 'False'; ExternalVisible := 'False'; ExternalWritable := 'False'} : "UDT_PECConfiguration";
         MCO_M01 { ExternalAccessible := 'False'; ExternalVisible := 'False'; ExternalWritable := 'False'} : "UDT_AixPlcFullControllerConfiguration";
      END_STRUCT;
      "490" { ExternalAccessible := 'False'; ExternalVisible := 'False'; ExternalWritable := 'False'} : Struct
         Conveyor { ExternalAccessible := 'False'; ExternalVisible := 'False'; ExternalWritable := 'False'; S7_SetPoint := 'False'} : "UDT_ConveyorConfiguration";
         PEC_EoS { ExternalAccessible := 'False'; ExternalVisible := 'False'; ExternalWritable := 'False'} : "UDT_PECConfiguration";
         MCO_M01 { ExternalAccessible := 'False'; ExternalVisible := 'False'; ExternalWritable := 'False'} : "UDT_AixPlcFullControllerConfiguration";
      END_STRUCT;
      "491" { ExternalAccessible := 'False'; ExternalVisible := 'False'; ExternalWritable := 'False'} : Struct
         Conveyor { ExternalAccessible := 'False'; ExternalVisible := 'False'; ExternalWritable := 'False'; S7_SetPoint := 'False'} : "UDT_ConveyorConfiguration";
         RightAngledTransfer { ExternalAccessible := 'False'; ExternalVisible := 'False'; ExternalWritable := 'False'; S7_SetPoint := 'False'} : "UDT_RATConfiguration";
         MCO_M01 { ExternalAccessible := 'False'; ExternalVisible := 'False'; ExternalWritable := 'False'} : "UDT_AixPlcFullControllerConfiguration";
      END_STRUCT;
      "500" { ExternalAccessible := 'False'; ExternalVisible := 'False'; ExternalWritable := 'False'} : Struct
         Conveyor { ExternalAccessible := 'False'; ExternalVisible := 'False'; ExternalWritable := 'False'; S7_SetPoint := 'False'} : "UDT_ConveyorConfiguration";
         PEC_EoS { ExternalAccessible := 'False'; ExternalVisible := 'False'; ExternalWritable := 'False'} : "UDT_PECConfiguration";
         MCO_M01 { ExternalAccessible := 'False'; ExternalVisible := 'False'; ExternalWritable := 'False'} : "UDT_AixPlcFullControllerConfiguration";
      END_STRUCT;
      "610" { ExternalAccessible := 'False'; ExternalVisible := 'False'; ExternalWritable := 'False'} : Struct
         Conveyor { ExternalAccessible := 'False'; ExternalVisible := 'False'; ExternalWritable := 'False'; S7_SetPoint := 'False'} : "UDT_ConveyorConfiguration";
         PEC_EoS { ExternalAccessible := 'False'; ExternalVisible := 'False'; ExternalWritable := 'False'} : "UDT_PECConfiguration";
         MCO_M01 { ExternalAccessible := 'False'; ExternalVisible := 'False'; ExternalWritable := 'False'} : "UDT_AixPlcFullControllerConfiguration";
      END_STRUCT;
      "611" { ExternalAccessible := 'False'; ExternalVisible := 'False'; ExternalWritable := 'False'} : Struct
         Conveyor { ExternalAccessible := 'False'; ExternalVisible := 'False'; ExternalWritable := 'False'; S7_SetPoint := 'False'} : "UDT_ConveyorConfiguration";
         RightAngledTransfer { ExternalAccessible := 'False'; ExternalVisible := 'False'; ExternalWritable := 'False'; S7_SetPoint := 'False'} : "UDT_RATConfiguration";
         MCO_M01 { ExternalAccessible := 'False'; ExternalVisible := 'False'; ExternalWritable := 'False'} : "UDT_AixPlcFullControllerConfiguration";
      END_STRUCT;
      "620" { ExternalAccessible := 'False'; ExternalVisible := 'False'; ExternalWritable := 'False'} : Struct
         Conveyor { ExternalAccessible := 'False'; ExternalVisible := 'False'; ExternalWritable := 'False'; S7_SetPoint := 'False'} : "UDT_ConveyorConfiguration";
         MCO_M01 { ExternalAccessible := 'False'; ExternalVisible := 'False'; ExternalWritable := 'False'} : "UDT_AixPlcFullControllerConfiguration";
      END_STRUCT;
      "630" { ExternalAccessible := 'False'; ExternalVisible := 'False'; ExternalWritable := 'False'} : Struct
         Conveyor { ExternalAccessible := 'False'; ExternalVisible := 'False'; ExternalWritable := 'False'; S7_SetPoint := 'False'} : "UDT_ConveyorConfiguration";
         MCO_M01 { ExternalAccessible := 'False'; ExternalVisible := 'False'; ExternalWritable := 'False'} : "UDT_AixPlcFullControllerConfiguration";
      END_STRUCT;
      "640" { ExternalAccessible := 'False'; ExternalVisible := 'False'; ExternalWritable := 'False'} : Struct
         Conveyor { ExternalAccessible := 'False'; ExternalVisible := 'False'; ExternalWritable := 'False'; S7_SetPoint := 'False'} : "UDT_ConveyorConfiguration";
         PEC_EoS { ExternalAccessible := 'False'; ExternalVisible := 'False'; ExternalWritable := 'False'} : "UDT_PECConfiguration";
         MCO_M01 { ExternalAccessible := 'False'; ExternalVisible := 'False'; ExternalWritable := 'False'} : "UDT_AixPlcFullControllerConfiguration";
      END_STRUCT;
   END_STRUCT;

END_TYPE

